LIN {X 0,Y 573.283,Z 141.077,A -85,B 0,C 180,E1 -2348.459,E2 -2348.459} C_VEL
LIN {X 0,Y 573.149,Z 141.164,A -85,B 0,C 180,E1 -2350.598,E2 -2350.598} C_VEL
LIN {X 0,Y 573.117,Z 144.62,A -85,B 0,C 180,E1 -2353.473,E2 -2353.473} C_VEL
LIN {X 0,Y 573.106,Z 148.053,A -85,B 0,C 180,E1 -2356.382,E2 -2356.382} C_VEL
LIN {X 0,Y 573.053,Z 151.315,A -85,B 0,C 180,E1 -2359.206,E2 -2359.206} C_VEL
LIN {X 0,Y 573.008,Z 154.185,A -85,B 0,C 180,E1 -2361.589,E2 -2361.589} C_VEL
LIN {X 0,Y 572.973,Z 157.111,A -85,B 0,C 180,E1 -2364.257,E2 -2364.257} C_VEL
LIN {X 0,Y 572.315,Z 157.815,A -85,B 0,C 180,E1 -2364.839,E2 -2364.839} C_VEL
LIN {X 0,Y 569.431,Z 159.133,A -85,B 0,C 180,E1 -2365.781,E2 -2365.781} C_VEL
LIN {X 0,Y 566.994,Z 160.207,A -85,B 0,C 180,E1 -2366.539,E2 -2366.539} C_VEL
LIN {X 0,Y 565.964,Z 160.962,A -85,B 0,C 180,E1 -2367.126,E2 -2367.126} C_VEL
LIN {X 0,Y 565.89,Z 161.194,A -85,B 0,C 180,E1 -2367.324,E2 -2367.324} C_VEL
LIN {X 0,Y 565.87,Z 164.215,A -85,B 0,C 180,E1 -2369.788,E2 -2369.788} C_VEL
LIN {X 0,Y 565.856,Z 167.674,A -85,B 0,C 180,E1 -2372.426,E2 -2372.426} C_VEL
LIN {X 0,Y 566.893,Z 175.191,A -85,B 0,C 180,E1 -2372.627,E2 -2372.627} C_VEL
LIN {X 0,Y 566.781,Z 187.823,A -85,B 0,C 180,E1 -2373.014,E2 -2373.014} C_VEL
LIN {X 0,Y 566.62,Z 199.261,A -85,B 0,C 180,E1 -2373.5,E2 -2373.5} C_VEL
LIN {X 0,Y 566.449,Z 210.991,A -85,B 0,C 180,E1 -2374.154,E2 -2374.154} C_VEL
LIN {X 0,Y 566.378,Z 222.253,A -85,B 0,C 180,E1 -2374.95,E2 -2374.95} C_VEL
LIN {X 0,Y 566.268,Z 230.723,A -85,B 0,C 180,E1 -2375.684,E2 -2375.684} C_VEL
LIN {X 0,Y 566.138,Z 239.28,A -85,B 0,C 180,E1 -2376.574,E2 -2376.574} C_VEL
LIN {X 0,Y 566.049,Z 247.98,A -85,B 0,C 180,E1 -2377.696,E2 -2377.696} C_VEL
LIN {X 0,Y 565.981,Z 255.315,A -85,B 0,C 180,E1 -2378.885,E2 -2378.885} C_VEL
LIN {X 0,Y 565.935,Z 260.327,A -85,B 0,C 180,E1 -2379.914,E2 -2379.914} C_VEL
LIN {X 0,Y 565.904,Z 264.999,A -85,B 0,C 180,E1 -2381.163,E2 -2381.163} C_VEL
LIN {X 0,Y 565.919,Z 267.606,A -85,B 0,C 180,E1 -2382.114,E2 -2382.114} C_VEL
LIN {X 0,Y 565.855,Z 269.477,A -85,B 0,C 180,E1 -2383.086,E2 -2383.086} C_VEL
LIN {X 0,Y 565.851,Z 270.609,A -85,B 0,C 180,E1 -2384.069,E2 -2384.069} C_VEL
LIN {X 0,Y 565.831,Z 270.999,A -85,B 0,C 180,E1 -2385.07,E2 -2385.07} C_VEL
LIN {X 0,Y 565.849,Z 270.565,A -85,B 0,C 180,E1 -2386.085,E2 -2386.085} C_VEL
LIN {X 0,Y 565.857,Z 269.292,A -85,B 0,C 180,E1 -2387.12,E2 -2387.12} C_VEL
LIN {X 0,Y 565.914,Z 267.122,A -85,B 0,C 180,E1 -2388.17,E2 -2388.17} C_VEL
LIN {X 0,Y 565.918,Z 263.923,A -85,B 0,C 180,E1 -2389.247,E2 -2389.247} C_VEL
LIN {X 0,Y 565.967,Z 259.569,A -85,B 0,C 180,E1 -2390.344,E2 -2390.344} C_VEL
LIN {X 0,Y 565.99,Z 253.825,A -85,B 0,C 180,E1 -2391.469,E2 -2391.469} C_VEL
LIN {X 0,Y 566.059,Z 246.426,A -85,B 0,C 180,E1 -2392.617,E2 -2392.617} C_VEL
LIN {X 0,Y 566.167,Z 238.204,A -85,B 0,C 180,E1 -2393.635,E2 -2393.635} C_VEL
LIN {X 0,Y 566.288,Z 229.712,A -85,B 0,C 180,E1 -2394.499,E2 -2394.499} C_VEL
LIN {X 0,Y 566.367,Z 220.17,A -85,B 0,C 180,E1 -2395.301,E2 -2395.301} C_VEL
LIN {X 0,Y 566.511,Z 208.941,A -85,B 0,C 180,E1 -2396.064,E2 -2396.064} C_VEL
LIN {X 0,Y 566.621,Z 197.802,A -85,B 0,C 180,E1 -2396.659,E2 -2396.659} C_VEL
LIN {X 0,Y 566.796,Z 186.076,A -85,B 0,C 180,E1 -2397.137,E2 -2397.137} C_VEL
LIN {X 0,Y 566.771,Z 173.284,A -85,B 0,C 180,E1 -2397.514,E2 -2397.514} C_VEL
LIN {X 0,Y 565.851,Z 167.7,A -85,B 0,C 180,E1 -2397.652,E2 -2397.652} C_VEL
LIN {X 0,Y 565.875,Z 164.107,A -85,B 0,C 180,E1 -2400.386,E2 -2400.386} C_VEL
LIN {X 0,Y 565.899,Z 160.384,A -85,B 0,C 180,E1 -2403.402,E2 -2403.402} C_VEL
LIN {X 0,Y 565.889,Z 157.605,A -85,B 0,C 180,E1 -2405.805,E2 -2405.805} C_VEL
LIN {X 0,Y 565.923,Z 154.307,A -85,B 0,C 180,E1 -2408.652,E2 -2408.652} C_VEL
LIN {X 0,Y 565.967,Z 151.289,A -85,B 0,C 180,E1 -2411.164,E2 -2411.164} C_VEL
LIN {X 0,Y 566.017,Z 148.71,A -85,B 0,C 180,E1 -2413.406,E2 -2413.406} C_VEL
LIN {X 0,Y 566.011,Z 145.176,A -85,B 0,C 180,E1 -2416.354,E2 -2416.354} C_VEL
LIN {X 0,Y 566.106,Z 142.346,A -85,B 0,C 180,E1 -2418.739,E2 -2418.739} C_VEL
LIN {X 0,Y 566.08,Z 141.976,A -85,B 0,C 180,E1 -2419.267,E2 -2419.267} C_VEL
LIN {X 0,Y 566.22,Z 141.957,A -85,B 0,C 180,E1 -2421.434,E2 -2421.434} C_VEL
LIN {X 0,Y 566.26,Z 141.951,A -85,B 0,C 180,E1 -2424.302,E2 -2424.302} C_VEL
LIN {X 0,Y 566.284,Z 141.948,A -85,B 0,C 180,E1 -2427.866,E2 -2427.866} C_VEL
LIN {X 0,Y 566.296,Z 141.946,A -85,B 0,C 180,E1 -2430.711,E2 -2430.711} C_VEL
LIN {X 0,Y 566.268,Z 141.949,A -85,B 0,C 180,E1 -2432.845,E2 -2432.845} C_VEL
LIN {X 0,Y 566.258,Z 141.951,A -85,B 0,C 180,E1 -2435.698,E2 -2435.698} C_VEL
LIN {X 0,Y 566.226,Z 141.956,A -85,B 0,C 180,E1 -2438.566,E2 -2438.566} C_VEL
LIN {X 0,Y 566.239,Z 141.953,A -85,B 0,C 180,E1 -2441.454,E2 -2441.454} C_VEL
LIN {X 0,Y 566.232,Z 141.956,A -85,B 0,C 180,E1 -2444.507,E2 -2444.507} C_VEL
LIN {X 0,Y 566.2,Z 141.958,A -85,B 0,C 180,E1 -2447.332,E2 -2447.332} C_VEL
LIN {X 0,Y 566.212,Z 141.958,A -85,B 0,C 180,E1 -2450.337,E2 -2450.337} C_VEL
LIN {X 0,Y 566.188,Z 141.959,A -85,B 0,C 180,E1 -2453.404,E2 -2453.404} C_VEL
LIN {X 0,Y 566.21,Z 141.957,A -85,B 0,C 180,E1 -2455.749,E2 -2455.749} C_VEL
LIN {X 0,Y 566.2,Z 141.957,A -85,B 0,C 180,E1 -2458.202,E2 -2458.202} C_VEL
LIN {X 0,Y 566.191,Z 141.96,A -85,B 0,C 180,E1 -2461.077,E2 -2461.077} C_VEL
LIN {X 0,Y 566.209,Z 141.96,A -85,B 0,C 180,E1 -2463.734,E2 -2463.734} C_VEL
LIN {X 0,Y 566.197,Z 141.958,A -85,B 0,C 180,E1 -2466.57,E2 -2466.57} C_VEL
LIN {X 0,Y 566.221,Z 141.955,A -85,B 0,C 180,E1 -2469.273,E2 -2469.273} C_VEL
LIN {X 0,Y 566.209,Z 141.959,A -85,B 0,C 180,E1 -2472.088,E2 -2472.088} C_VEL
LIN {X 0,Y 566.171,Z 141.962,A -85,B 0,C 180,E1 -2475.036,E2 -2475.036} C_VEL
LIN {X 0,Y 566.187,Z 141.96,A -85,B 0,C 180,E1 -2477.911,E2 -2477.911} C_VEL
LIN {X 0,Y 566.216,Z 141.959,A -85,B 0,C 180,E1 -2480.727,E2 -2480.727} C_VEL
LIN {X 0,Y 566.2,Z 141.957,A -85,B 0,C 180,E1 -2483.786,E2 -2483.786} C_VEL
LIN {X 0,Y 566.197,Z 141.958,A -85,B 0,C 180,E1 -2486.268,E2 -2486.268} C_VEL
LIN {X 0,Y 566.193,Z 141.96,A -85,B 0,C 180,E1 -2488.924,E2 -2488.924} C_VEL
LIN {X 0,Y 566.211,Z 141.957,A -85,B 0,C 180,E1 -2491.858,E2 -2491.858} C_VEL
LIN {X 0,Y 566.214,Z 141.957,A -85,B 0,C 180,E1 -2494.251,E2 -2494.251} C_VEL
LIN {X 0,Y 566.171,Z 141.962,A -85,B 0,C 180,E1 -2496.719,E2 -2496.719} C_VEL
LIN {X 0,Y 566.212,Z 141.956,A -85,B 0,C 180,E1 -2499.663,E2 -2499.663} C_VEL
LIN {X 0,Y 566.197,Z 141.959,A -85,B 0,C 180,E1 -2502.669,E2 -2502.669} C_VEL
LIN {X 0,Y 566.222,Z 141.955,A -85,B 0,C 180,E1 -2505.627,E2 -2505.627} C_VEL
LIN {X 0,Y 566.236,Z 141.954,A -85,B 0,C 180,E1 -2508.676,E2 -2508.676} C_VEL
LIN {X 0,Y 566.208,Z 141.956,A -85,B 0,C 180,E1 -2511.434,E2 -2511.434} C_VEL
LIN {X 0,Y 566.26,Z 141.952,A -85,B 0,C 180,E1 -2514.302,E2 -2514.302} C_VEL
LIN {X 0,Y 566.285,Z 141.948,A -85,B 0,C 180,E1 -2517.867,E2 -2517.867} C_VEL
LIN {X 0,Y 566.303,Z 141.946,A -85,B 0,C 180,E1 -2520.711,E2 -2520.711} C_VEL
LIN {X 0,Y 566.272,Z 141.952,A -85,B 0,C 180,E1 -2522.846,E2 -2522.846} C_VEL
LIN {X 0,Y 566.264,Z 141.95,A -85,B 0,C 180,E1 -2525.699,E2 -2525.699} C_VEL
LIN {X 0,Y 566.208,Z 141.957,A -85,B 0,C 180,E1 -2528.566,E2 -2528.566} C_VEL
LIN {X 0,Y 566.245,Z 141.955,A -85,B 0,C 180,E1 -2531.455,E2 -2531.455} C_VEL
LIN {X 0,Y 566.225,Z 141.954,A -85,B 0,C 180,E1 -2534.502,E2 -2534.502} C_VEL
LIN {X 0,Y 566.202,Z 141.96,A -85,B 0,C 180,E1 -2537.332,E2 -2537.332} C_VEL
LIN {X 0,Y 566.208,Z 141.956,A -85,B 0,C 180,E1 -2540.338,E2 -2540.338} C_VEL
LIN {X 0,Y 566.169,Z 141.963,A -85,B 0,C 180,E1 -2543.28,E2 -2543.28} C_VEL
LIN {X 0,Y 566.217,Z 141.958,A -85,B 0,C 180,E1 -2545.749,E2 -2545.749} C_VEL
LIN {X 0,Y 566.206,Z 141.96,A -85,B 0,C 180,E1 -2548.202,E2 -2548.202} C_VEL
LIN {X 0,Y 566.195,Z 141.959,A -85,B 0,C 180,E1 -2551.077,E2 -2551.077} C_VEL
LIN {X 0,Y 566.199,Z 141.958,A -85,B 0,C 180,E1 -2553.732,E2 -2553.732} C_VEL
LIN {X 0,Y 566.202,Z 141.959,A -85,B 0,C 180,E1 -2556.57,E2 -2556.57} C_VEL
LIN {X 0,Y 566.216,Z 141.955,A -85,B 0,C 180,E1 -2559.686,E2 -2559.686} C_VEL
LIN {X 0,Y 566.204,Z 141.958,A -85,B 0,C 180,E1 -2562.917,E2 -2562.917} C_VEL
LIN {X 0,Y 566.197,Z 141.957,A -85,B 0,C 180,E1 -2566.049,E2 -2566.049} C_VEL
LIN {X 0,Y 566.206,Z 141.957,A -85,B 0,C 180,E1 -2569.215,E2 -2569.215} C_VEL
LIN {X 0,Y 566.188,Z 141.961,A -85,B 0,C 180,E1 -2571.637,E2 -2571.637} C_VEL
LIN {X 0,Y 566.237,Z 141.963,A -85,B 0,C 180,E1 -2572.989,E2 -2572.989} C_VEL
LIN {X 0,Y 566.793,Z 145.917,A -85,B 0,C 180,E1 -2574.354,E2 -2574.354} C_VEL
LIN {X 0,Y 566.8,Z 152.68,A -85,B 0,C 180,E1 -2576.557,E2 -2576.557} C_VEL
LIN {X 0,Y 566.62,Z 161.803,A -85,B 0,C 180,E1 -2579.433,E2 -2579.433} C_VEL
LIN {X 0,Y 566.518,Z 171.071,A -85,B 0,C 180,E1 -2582.276,E2 -2582.276} C_VEL
LIN {X 0,Y 566.418,Z 180.338,A -85,B 0,C 180,E1 -2585.048,E2 -2585.048} C_VEL
LIN {X 0,Y 566.323,Z 190.929,A -85,B 0,C 180,E1 -2588.143,E2 -2588.143} C_VEL
LIN {X 0,Y 566.186,Z 201.521,A -85,B 0,C 180,E1 -2591.172,E2 -2591.172} C_VEL
LIN {X 0,Y 566.112,Z 212.112,A -85,B 0,C 180,E1 -2594.15,E2 -2594.15} C_VEL
LIN {X 0,Y 566.003,Z 222.703,A -85,B 0,C 180,E1 -2597.085,E2 -2597.085} C_VEL
LIN {X 0,Y 566.011,Z 223.53,A -85,B 0,C 180,E1 -2597.313,E2 -2597.313} C_VEL
LIN {X 0,Y 566.93,Z 230.375,A -85,B 0,C 180,E1 -2597.471,E2 -2597.471} C_VEL
LIN {X 0,Y 566.839,Z 242.5,A -85,B 0,C 180,E1 -2597.787,E2 -2597.787} C_VEL
LIN {X 0,Y 566.68,Z 254.321,A -85,B 0,C 180,E1 -2598.228,E2 -2598.228} C_VEL
LIN {X 0,Y 566.532,Z 266.981,A -85,B 0,C 180,E1 -2598.868,E2 -2598.868} C_VEL
LIN {X 0,Y 566.434,Z 278.748,A -85,B 0,C 180,E1 -2599.636,E2 -2599.636} C_VEL
LIN {X 0,Y 566.301,Z 287.648,A -85,B 0,C 180,E1 -2600.355,E2 -2600.355} C_VEL
LIN {X 0,Y 566.166,Z 296.788,A -85,B 0,C 180,E1 -2601.254,E2 -2601.254} C_VEL
LIN {X 0,Y 566.081,Z 305.691,A -85,B 0,C 180,E1 -2602.33,E2 -2602.33} C_VEL
LIN {X 0,Y 565.968,Z 312.956,A -85,B 0,C 180,E1 -2603.422,E2 -2603.422} C_VEL
LIN {X 0,Y 566.004,Z 317.681,A -85,B 0,C 180,E1 -2604.299,E2 -2604.299} C_VEL
LIN {X 0,Y 565.933,Z 322.372,A -85,B 0,C 180,E1 -2605.37,E2 -2605.37} C_VEL
LIN {X 0,Y 565.927,Z 325.957,A -85,B 0,C 180,E1 -2606.44,E2 -2606.44} C_VEL
LIN {X 0,Y 565.878,Z 327.809,A -85,B 0,C 180,E1 -2607.153,E2 -2607.153} C_VEL
LIN {X 0,Y 565.841,Z 329.2,A -85,B 0,C 180,E1 -2607.865,E2 -2607.865} C_VEL
LIN {X 0,Y 565.841,Z 330.784,A -85,B 0,C 180,E1 -2609.288,E2 -2609.288} C_VEL
LIN {X 0,Y 565.839,Z 331,A -85,B 0,C 180,E1 -2610,E2 -2610} C_VEL
LIN {X 0,Y 565.846,Z 330.185,A -85,B 0,C 180,E1 -2611.424,E2 -2611.424} C_VEL
LIN {X 0,Y 565.841,Z 329.201,A -85,B 0,C 180,E1 -2612.136,E2 -2612.136} C_VEL
LIN {X 0,Y 565.878,Z 327.809,A -85,B 0,C 180,E1 -2612.848,E2 -2612.848} C_VEL
LIN {X 0,Y 565.926,Z 324.896,A -85,B 0,C 180,E1 -2613.917,E2 -2613.917} C_VEL
LIN {X 0,Y 565.878,Z 320.949,A -85,B 0,C 180,E1 -2614.988,E2 -2614.988} C_VEL
LIN {X 0,Y 566.002,Z 315.866,A -85,B 0,C 180,E1 -2616.059,E2 -2616.059} C_VEL
LIN {X 0,Y 566.041,Z 309.469,A -85,B 0,C 180,E1 -2617.132,E2 -2617.132} C_VEL
LIN {X 0,Y 566.134,Z 301.477,A -85,B 0,C 180,E1 -2618.208,E2 -2618.208} C_VEL
LIN {X 0,Y 566.229,Z 293.335,A -85,B 0,C 180,E1 -2619.106,E2 -2619.106} C_VEL
LIN {X 0,Y 566.344,Z 283.4,A -85,B 0,C 180,E1 -2620.005,E2 -2620.005} C_VEL
LIN {X 0,Y 566.501,Z 272.326,A -85,B 0,C 180,E1 -2620.805,E2 -2620.805} C_VEL
LIN {X 0,Y 566.574,Z 261.175,A -85,B 0,C 180,E1 -2621.448,E2 -2621.448} C_VEL
LIN {X 0,Y 566.741,Z 248.985,A -85,B 0,C 180,E1 -2621.988,E2 -2621.988} C_VEL
LIN {X 0,Y 566.918,Z 236.171,A -85,B 0,C 180,E1 -2622.393,E2 -2622.393} C_VEL
LIN {X 0,Y 566.73,Z 228.079,A -85,B 0,C 180,E1 -2622.58,E2 -2622.58} C_VEL
LIN {X 0,Y 566.011,Z 223.53,A -85,B 0,C 180,E1 -2622.687,E2 -2622.687} C_VEL
LIN {X 0,Y 566.087,Z 213.435,A -85,B 0,C 180,E1 -2625.481,E2 -2625.481} C_VEL
LIN {X 0,Y 566.167,Z 202.844,A -85,B 0,C 180,E1 -2628.454,E2 -2628.454} C_VEL
LIN {X 0,Y 566.246,Z 193.576,A -85,B 0,C 180,E1 -2631.096,E2 -2631.096} C_VEL
LIN {X 0,Y 566.365,Z 184.309,A -85,B 0,C 180,E1 -2633.784,E2 -2633.784} C_VEL
LIN {X 0,Y 566.485,Z 175.042,A -85,B 0,C 180,E1 -2636.528,E2 -2636.528} C_VEL
LIN {X 0,Y 566.553,Z 165.774,A -85,B 0,C 180,E1 -2639.34,E2 -2639.34} C_VEL
LIN {X 0,Y 566.704,Z 156.507,A -85,B 0,C 180,E1 -2642.227,E2 -2642.227} C_VEL
LIN {X 0,Y 566.837,Z 148.564,A -85,B 0,C 180,E1 -2644.774,E2 -2644.774} C_VEL
LIN {X 0,Y 566.568,Z 144.069,A -85,B 0,C 180,E1 -2646.264,E2 -2646.264} C_VEL
LIN {X 0,Y 566.239,Z 141.957,A -85,B 0,C 180,E1 -2647.011,E2 -2647.011} C_VEL
LIN {X 0,Y 566.22,Z 141.957,A -85,B 0,C 180,E1 -2649.686,E2 -2649.686} C_VEL
LIN {X 0,Y 566.216,Z 141.959,A -85,B 0,C 180,E1 -2652.088,E2 -2652.088} C_VEL
LIN {X 0,Y 566.178,Z 141.963,A -85,B 0,C 180,E1 -2655.036,E2 -2655.036} C_VEL
LIN {X 0,Y 566.194,Z 141.961,A -85,B 0,C 180,E1 -2657.91,E2 -2657.91} C_VEL
LIN {X 0,Y 566.225,Z 141.956,A -85,B 0,C 180,E1 -2660.727,E2 -2660.727} C_VEL
LIN {X 0,Y 566.19,Z 141.96,A -85,B 0,C 180,E1 -2663.788,E2 -2663.788} C_VEL
LIN {X 0,Y 566.217,Z 141.958,A -85,B 0,C 180,E1 -2666.266,E2 -2666.266} C_VEL
LIN {X 0,Y 566.199,Z 141.959,A -85,B 0,C 180,E1 -2668.923,E2 -2668.923} C_VEL
LIN {X 0,Y 566.217,Z 141.957,A -85,B 0,C 180,E1 -2671.857,E2 -2671.857} C_VEL
LIN {X 0,Y 566.219,Z 141.957,A -85,B 0,C 180,E1 -2674.251,E2 -2674.251} C_VEL
LIN {X 0,Y 566.176,Z 141.962,A -85,B 0,C 180,E1 -2676.719,E2 -2676.719} C_VEL
LIN {X 0,Y 566.212,Z 141.958,A -85,B 0,C 180,E1 -2679.662,E2 -2679.662} C_VEL
LIN {X 0,Y 566.204,Z 141.959,A -85,B 0,C 180,E1 -2682.668,E2 -2682.668} C_VEL
LIN {X 0,Y 566.24,Z 141.955,A -85,B 0,C 180,E1 -2685.627,E2 -2685.627} C_VEL
LIN {X 0,Y 566.24,Z 141.955,A -85,B 0,C 180,E1 -2688.675,E2 -2688.675} C_VEL
LIN {X 0,Y 566.233,Z 141.956,A -85,B 0,C 180,E1 -2691.434,E2 -2691.434} C_VEL
LIN {X 0,Y 566.265,Z 141.951,A -85,B 0,C 180,E1 -2694.301,E2 -2694.301} C_VEL
LIN {X 0,Y 566.288,Z 141.949,A -85,B 0,C 180,E1 -2697.866,E2 -2697.866} C_VEL
LIN {X 0,Y 566.308,Z 141.947,A -85,B 0,C 180,E1 -2700.711,E2 -2700.711} C_VEL
LIN {X 0,Y 566.276,Z 141.951,A -85,B 0,C 180,E1 -2702.845,E2 -2702.845} C_VEL
LIN {X 0,Y 566.26,Z 141.954,A -85,B 0,C 180,E1 -2705.698,E2 -2705.698} C_VEL
LIN {X 0,Y 566.225,Z 141.957,A -85,B 0,C 180,E1 -2708.565,E2 -2708.565} C_VEL
LIN {X 0,Y 566.082,Z 142.035,A -85,B 0,C 180,E1 -2710.732,E2 -2710.732} C_VEL
LIN {X 0,Y 566.051,Z 145.513,A -85,B 0,C 180,E1 -2713.644,E2 -2713.644} C_VEL
LIN {X 0,Y 566.047,Z 148.957,A -85,B 0,C 180,E1 -2716.592,E2 -2716.592} C_VEL
LIN {X 0,Y 565.936,Z 152.413,A -85,B 0,C 180,E1 -2719.59,E2 -2719.59} C_VEL
LIN {X 0,Y 565.916,Z 155.096,A -85,B 0,C 180,E1 -2721.873,E2 -2721.873} C_VEL
LIN {X 0,Y 565.903,Z 157.781,A -85,B 0,C 180,E1 -2724.248,E2 -2724.248} C_VEL
LIN {X 0,Y 565.903,Z 160.372,A -85,B 0,C 180,E1 -2726.597,E2 -2726.597} C_VEL
LIN {X 0,Y 565.89,Z 161.194,A -85,B 0,C 180,E1 -2727.324,E2 -2727.324} C_VEL
LIN {X 0,Y 565.244,Z 161.922,A -85,B 0,C 180,E1 -2727.914,E2 -2727.914} C_VEL
LIN {X 0,Y 562.374,Z 163.269,A -85,B 0,C 180,E1 -2728.869,E2 -2728.869} C_VEL
LIN {X 0,Y 559.925,Z 164.365,A -85,B 0,C 180,E1 -2729.637,E2 -2729.637} C_VEL
LIN {X 0,Y 558.86,Z 165.144,A -85,B 0,C 180,E1 -2730.231,E2 -2730.231} C_VEL
LIN {X 0,Y 558.767,Z 165.387,A -85,B 0,C 180,E1 -2730.433,E2 -2730.433} C_VEL
LIN {X 0,Y 558.759,Z 167.671,A -85,B 0,C 180,E1 -2732.26,E2 -2732.26} C_VEL
LIN {X 0,Y 559.961,Z 175.931,A -85,B 0,C 180,E1 -2732.489,E2 -2732.489} C_VEL
LIN {X 0,Y 559.827,Z 188.735,A -85,B 0,C 180,E1 -2732.897,E2 -2732.897} C_VEL
LIN {X 0,Y 559.621,Z 200.62,A -85,B 0,C 180,E1 -2733.425,E2 -2733.425} C_VEL
LIN {X 0,Y 559.462,Z 212.087,A -85,B 0,C 180,E1 -2734.087,E2 -2734.087} C_VEL
LIN {X 0,Y 559.356,Z 222.83,A -85,B 0,C 180,E1 -2734.867,E2 -2734.867} C_VEL
LIN {X 0,Y 559.206,Z 232.71,A -85,B 0,C 180,E1 -2735.76,E2 -2735.76} C_VEL
LIN {X 0,Y 559.069,Z 241.597,A -85,B 0,C 180,E1 -2736.748,E2 -2736.748} C_VEL
LIN {X 0,Y 558.96,Z 249.3,A -85,B 0,C 180,E1 -2737.797,E2 -2737.797} C_VEL
LIN {X 0,Y 558.896,Z 256.106,A -85,B 0,C 180,E1 -2738.957,E2 -2738.957} C_VEL
LIN {X 0,Y 558.859,Z 260.573,A -85,B 0,C 180,E1 -2739.904,E2 -2739.904} C_VEL
LIN {X 0,Y 558.81,Z 264.676,A -85,B 0,C 180,E1 -2741.009,E2 -2741.009} C_VEL
LIN {X 0,Y 558.82,Z 267.655,A -85,B 0,C 180,E1 -2742.096,E2 -2742.096} C_VEL
LIN {X 0,Y 558.767,Z 269.62,A -85,B 0,C 180,E1 -2743.155,E2 -2743.155} C_VEL
LIN {X 0,Y 558.765,Z 270.703,A -85,B 0,C 180,E1 -2744.198,E2 -2744.198} C_VEL
LIN {X 0,Y 558.75,Z 270.968,A -85,B 0,C 180,E1 -2745.221,E2 -2745.221} C_VEL
LIN {X 0,Y 558.758,Z 270.465,A -85,B 0,C 180,E1 -2746.228,E2 -2746.228} C_VEL
LIN {X 0,Y 558.759,Z 269.178,A -85,B 0,C 180,E1 -2747.218,E2 -2747.218} C_VEL
LIN {X 0,Y 558.815,Z 267.151,A -85,B 0,C 180,E1 -2748.197,E2 -2748.197} C_VEL
LIN {X 0,Y 558.822,Z 264.414,A -85,B 0,C 180,E1 -2749.158,E2 -2749.158} C_VEL
LIN {X 0,Y 558.881,Z 259.874,A -85,B 0,C 180,E1 -2750.343,E2 -2750.343} C_VEL
LIN {X 0,Y 558.925,Z 253.564,A -85,B 0,C 180,E1 -2751.598,E2 -2751.598} C_VEL
LIN {X 0,Y 558.985,Z 246.996,A -85,B 0,C 180,E1 -2752.632,E2 -2752.632} C_VEL
LIN {X 0,Y 559.084,Z 239.797,A -85,B 0,C 180,E1 -2753.563,E2 -2753.563} C_VEL
LIN {X 0,Y 559.262,Z 230.183,A -85,B 0,C 180,E1 -2754.575,E2 -2754.575} C_VEL
LIN {X 0,Y 559.392,Z 219.751,A -85,B 0,C 180,E1 -2755.463,E2 -2755.463} C_VEL
LIN {X 0,Y 559.526,Z 208.818,A -85,B 0,C 180,E1 -2756.211,E2 -2756.211} C_VEL
LIN {X 0,Y 559.687,Z 197.086,A -85,B 0,C 180,E1 -2756.838,E2 -2756.838} C_VEL
LIN {X 0,Y 559.874,Z 184.86,A -85,B 0,C 180,E1 -2757.332,E2 -2757.332} C_VEL
LIN {X 0,Y 559.794,Z 173.908,A -85,B 0,C 180,E1 -2757.656,E2 -2757.656} C_VEL
LIN {X 0,Y 558.763,Z 167.684,A -85,B 0,C 180,E1 -2757.819,E2 -2757.819} C_VEL
LIN {X 0,Y 558.794,Z 164.191,A -85,B 0,C 180,E1 -2760.626,E2 -2760.626} C_VEL
LIN {X 0,Y 558.813,Z 160.368,A -85,B 0,C 180,E1 -2763.884,E2 -2763.884} C_VEL
LIN {X 0,Y 558.833,Z 157.24,A -85,B 0,C 180,E1 -2766.643,E2 -2766.643} C_VEL
LIN {X 0,Y 558.849,Z 153.987,A -85,B 0,C 180,E1 -2769.383,E2 -2769.383} C_VEL
LIN {X 0,Y 558.92,Z 150.432,A -85,B 0,C 180,E1 -2772.435,E2 -2772.435} C_VEL
LIN {X 0,Y 558.972,Z 146.812,A -85,B 0,C 180,E1 -2775.493,E2 -2775.493} C_VEL
LIN {X 0,Y 559.037,Z 143.059,A -85,B 0,C 180,E1 -2778.689,E2 -2778.689} C_VEL
LIN {X 0,Y 559.177,Z 142.834,A -85,B 0,C 180,E1 -2781.325,E2 -2781.325} C_VEL
LIN {X 0,Y 559.228,Z 142.827,A -85,B 0,C 180,E1 -2784.23,E2 -2784.23} C_VEL
LIN {X 0,Y 559.255,Z 142.824,A -85,B 0,C 180,E1 -2787.839,E2 -2787.839} C_VEL
LIN {X 0,Y 559.267,Z 142.821,A -85,B 0,C 180,E1 -2790.72,E2 -2790.72} C_VEL
LIN {X 0,Y 559.234,Z 142.824,A -85,B 0,C 180,E1 -2792.881,E2 -2792.881} C_VEL
LIN {X 0,Y 559.227,Z 142.828,A -85,B 0,C 180,E1 -2795.77,E2 -2795.77} C_VEL
LIN {X 0,Y 559.184,Z 142.832,A -85,B 0,C 180,E1 -2798.674,E2 -2798.674} C_VEL
LIN {X 0,Y 559.203,Z 142.83,A -85,B 0,C 180,E1 -2801.6,E2 -2801.6} C_VEL
LIN {X 0,Y 559.197,Z 142.832,A -85,B 0,C 180,E1 -2804.596,E2 -2804.596} C_VEL
LIN {X 0,Y 559.16,Z 142.835,A -85,B 0,C 180,E1 -2807.557,E2 -2807.557} C_VEL
LIN {X 0,Y 559.168,Z 142.834,A -85,B 0,C 180,E1 -2809.837,E2 -2809.837} C_VEL
LIN {X 0,Y 559.138,Z 142.837,A -85,B 0,C 180,E1 -2812.153,E2 -2812.153} C_VEL
LIN {X 0,Y 559.176,Z 142.834,A -85,B 0,C 180,E1 -2815.187,E2 -2815.187} C_VEL
LIN {X 0,Y 559.178,Z 142.836,A -85,B 0,C 180,E1 -2817.712,E2 -2817.712} C_VEL
LIN {X 0,Y 559.154,Z 142.838,A -85,B 0,C 180,E1 -2820.183,E2 -2820.183} C_VEL
LIN {X 0,Y 559.172,Z 142.835,A -85,B 0,C 180,E1 -2822.714,E2 -2822.714} C_VEL
LIN {X 0,Y 559.125,Z 142.84,A -85,B 0,C 180,E1 -2825.324,E2 -2825.324} C_VEL
LIN {X 0,Y 559.132,Z 142.837,A -85,B 0,C 180,E1 -2828.018,E2 -2828.018} C_VEL
LIN {X 0,Y 559.173,Z 142.834,A -85,B 0,C 180,E1 -2830.811,E2 -2830.811} C_VEL
LIN {X 0,Y 559.139,Z 142.837,A -85,B 0,C 180,E1 -2833.734,E2 -2833.734} C_VEL
LIN {X 0,Y 559.144,Z 142.838,A -85,B 0,C 180,E1 -2836.804,E2 -2836.804} C_VEL
LIN {X 0,Y 559.154,Z 142.837,A -85,B 0,C 180,E1 -2839.188,E2 -2839.188} C_VEL
LIN {X 0,Y 559.134,Z 142.84,A -85,B 0,C 180,E1 -2841.983,E2 -2841.983} C_VEL
LIN {X 0,Y 559.146,Z 142.837,A -85,B 0,C 180,E1 -2844.785,E2 -2844.785} C_VEL
LIN {X 0,Y 559.154,Z 142.835,A -85,B 0,C 180,E1 -2847.365,E2 -2847.365} C_VEL
LIN {X 0,Y 559.145,Z 142.837,A -85,B 0,C 180,E1 -2850.143,E2 -2850.143} C_VEL
LIN {X 0,Y 559.169,Z 142.834,A -85,B 0,C 180,E1 -2853.098,E2 -2853.098} C_VEL
LIN {X 0,Y 559.155,Z 142.835,A -85,B 0,C 180,E1 -2855.495,E2 -2855.495} C_VEL
LIN {X 0,Y 559.173,Z 142.835,A -85,B 0,C 180,E1 -2858.624,E2 -2858.624} C_VEL
LIN {X 0,Y 559.165,Z 142.835,A -85,B 0,C 180,E1 -2860.927,E2 -2860.927} C_VEL
LIN {X 0,Y 559.164,Z 142.835,A -85,B 0,C 180,E1 -2863.948,E2 -2863.948} C_VEL
LIN {X 0,Y 559.166,Z 142.836,A -85,B 0,C 180,E1 -2866.184,E2 -2866.184} C_VEL
LIN {X 0,Y 559.208,Z 142.83,A -85,B 0,C 180,E1 -2868.605,E2 -2868.605} C_VEL
LIN {X 0,Y 559.172,Z 142.833,A -85,B 0,C 180,E1 -2871.326,E2 -2871.326} C_VEL
LIN {X 0,Y 559.23,Z 142.827,A -85,B 0,C 180,E1 -2874.23,E2 -2874.23} C_VEL
LIN {X 0,Y 559.256,Z 142.824,A -85,B 0,C 180,E1 -2877.84,E2 -2877.84} C_VEL
LIN {X 0,Y 559.273,Z 142.821,A -85,B 0,C 180,E1 -2880.72,E2 -2880.72} C_VEL
LIN {X 0,Y 559.239,Z 142.827,A -85,B 0,C 180,E1 -2882.882,E2 -2882.882} C_VEL
LIN {X 0,Y 559.232,Z 142.826,A -85,B 0,C 180,E1 -2885.771,E2 -2885.771} C_VEL
LIN {X 0,Y 559.173,Z 142.834,A -85,B 0,C 180,E1 -2888.675,E2 -2888.675} C_VEL
LIN {X 0,Y 559.209,Z 142.83,A -85,B 0,C 180,E1 -2891.601,E2 -2891.601} C_VEL
LIN {X 0,Y 559.183,Z 142.832,A -85,B 0,C 180,E1 -2894.588,E2 -2894.588} C_VEL
LIN {X 0,Y 559.161,Z 142.837,A -85,B 0,C 180,E1 -2897.557,E2 -2897.557} C_VEL
LIN {X 0,Y 559.168,Z 142.837,A -85,B 0,C 180,E1 -2899.838,E2 -2899.838} C_VEL
LIN {X 0,Y 559.144,Z 142.84,A -85,B 0,C 180,E1 -2902.153,E2 -2902.153} C_VEL
LIN {X 0,Y 559.179,Z 142.832,A -85,B 0,C 180,E1 -2905.298,E2 -2905.298} C_VEL
LIN {X 0,Y 559.16,Z 142.835,A -85,B 0,C 180,E1 -2907.714,E2 -2907.714} C_VEL
LIN {X 0,Y 559.153,Z 142.835,A -85,B 0,C 180,E1 -2910.183,E2 -2910.183} C_VEL
LIN {X 0,Y 559.154,Z 142.835,A -85,B 0,C 180,E1 -2912.716,E2 -2912.716} C_VEL
LIN {X 0,Y 559.13,Z 142.84,A -85,B 0,C 180,E1 -2915.324,E2 -2915.324} C_VEL
LIN {X 0,Y 559.134,Z 142.84,A -85,B 0,C 180,E1 -2918.018,E2 -2918.018} C_VEL
LIN {X 0,Y 559.158,Z 142.835,A -85,B 0,C 180,E1 -2920.813,E2 -2920.813} C_VEL
LIN {X 0,Y 559.144,Z 142.837,A -85,B 0,C 180,E1 -2923.734,E2 -2923.734} C_VEL
LIN {X 0,Y 559.148,Z 142.835,A -85,B 0,C 180,E1 -2926.804,E2 -2926.804} C_VEL
LIN {X 0,Y 559.158,Z 142.836,A -85,B 0,C 180,E1 -2929.188,E2 -2929.188} C_VEL
LIN {X 0,Y 559.135,Z 142.84,A -85,B 0,C 180,E1 -2931.983,E2 -2931.983} C_VEL
LIN {X 0,Y 559.215,Z 143.016,A -85,B 0,C 180,E1 -2932.8,E2 -2932.8} C_VEL
LIN {X 0,Y 559.845,Z 147.254,A -85,B 0,C 180,E1 -2934.287,E2 -2934.287} C_VEL
LIN {X 0,Y 559.794,Z 155.185,A -85,B 0,C 180,E1 -2936.899,E2 -2936.899} C_VEL
LIN {X 0,Y 559.643,Z 164.451,A -85,B 0,C 180,E1 -2939.846,E2 -2939.846} C_VEL
LIN {X 0,Y 559.499,Z 173.719,A -85,B 0,C 180,E1 -2942.711,E2 -2942.711} C_VEL
LIN {X 0,Y 559.378,Z 182.986,A -85,B 0,C 180,E1 -2945.505,E2 -2945.505} C_VEL
LIN {X 0,Y 559.234,Z 193.577,A -85,B 0,C 180,E1 -2948.626,E2 -2948.626} C_VEL
LIN {X 0,Y 559.134,Z 202.844,A -85,B 0,C 180,E1 -2951.306,E2 -2951.306} C_VEL
LIN {X 0,Y 559.052,Z 213.436,A -85,B 0,C 180,E1 -2954.319,E2 -2954.319} C_VEL
LIN {X 0,Y 558.938,Z 223.53,A -85,B 0,C 180,E1 -2957.15,E2 -2957.15} C_VEL
LIN {X 0,Y 560.018,Z 231.514,A -85,B 0,C 180,E1 -2957.337,E2 -2957.337} C_VEL
LIN {X 0,Y 559.899,Z 243.88,A -85,B 0,C 180,E1 -2957.679,E2 -2957.679} C_VEL
LIN {X 0,Y 559.718,Z 256.284,A -85,B 0,C 180,E1 -2958.171,E2 -2958.171} C_VEL
LIN {X 0,Y 559.555,Z 267.767,A -85,B 0,C 180,E1 -2958.773,E2 -2958.773} C_VEL
LIN {X 0,Y 559.424,Z 278.748,A -85,B 0,C 180,E1 -2959.504,E2 -2959.504} C_VEL
LIN {X 0,Y 559.244,Z 289.602,A -85,B 0,C 180,E1 -2960.415,E2 -2960.415} C_VEL
LIN {X 0,Y 559.127,Z 298.414,A -85,B 0,C 180,E1 -2961.325,E2 -2961.325} C_VEL
LIN {X 0,Y 558.996,Z 307.001,A -85,B 0,C 180,E1 -2962.414,E2 -2962.414} C_VEL
LIN {X 0,Y 558.885,Z 314.689,A -85,B 0,C 180,E1 -2963.649,E2 -2963.649} C_VEL
LIN {X 0,Y 558.869,Z 319.366,A -85,B 0,C 180,E1 -2964.588,E2 -2964.588} C_VEL
LIN {X 0,Y 558.869,Z 323.678,A -85,B 0,C 180,E1 -2965.673,E2 -2965.673} C_VEL
LIN {X 0,Y 558.836,Z 325.957,A -85,B 0,C 180,E1 -2966.395,E2 -2966.395} C_VEL
LIN {X 0,Y 558.799,Z 327.809,A -85,B 0,C 180,E1 -2967.116,E2 -2967.116} C_VEL
LIN {X 0,Y 558.747,Z 329.2,A -85,B 0,C 180,E1 -2967.838,E2 -2967.838} C_VEL
LIN {X 0,Y 558.741,Z 330.785,A -85,B 0,C 180,E1 -2969.279,E2 -2969.279} C_VEL
LIN {X 0,Y 558.74,Z 331,A -85,B 0,C 180,E1 -2970,E2 -2970} C_VEL
LIN {X 0,Y 558.745,Z 330.185,A -85,B 0,C 180,E1 -2971.442,E2 -2971.442} C_VEL
LIN {X 0,Y 558.747,Z 329.2,A -85,B 0,C 180,E1 -2972.163,E2 -2972.163} C_VEL
LIN {X 0,Y 558.799,Z 327.809,A -85,B 0,C 180,E1 -2972.884,E2 -2972.884} C_VEL
LIN {X 0,Y 558.844,Z 324.895,A -85,B 0,C 180,E1 -2973.966,E2 -2973.966} C_VEL
LIN {X 0,Y 558.798,Z 320.949,A -85,B 0,C 180,E1 -2975.051,E2 -2975.051} C_VEL
LIN {X 0,Y 558.922,Z 315.866,A -85,B 0,C 180,E1 -2976.136,E2 -2976.136} C_VEL
LIN {X 0,Y 558.978,Z 309.468,A -85,B 0,C 180,E1 -2977.223,E2 -2977.223} C_VEL
LIN {X 0,Y 559.099,Z 301.477,A -85,B 0,C 180,E1 -2978.312,E2 -2978.312} C_VEL
LIN {X 0,Y 559.195,Z 293.335,A -85,B 0,C 180,E1 -2979.221,E2 -2979.221} C_VEL
LIN {X 0,Y 559.358,Z 283.4,A -85,B 0,C 180,E1 -2980.131,E2 -2980.131} C_VEL
LIN {X 0,Y 559.511,Z 272.435,A -85,B 0,C 180,E1 -2980.935,E2 -2980.935} C_VEL
LIN {X 0,Y 559.637,Z 260.82,A -85,B 0,C 180,E1 -2981.61,E2 -2981.61} C_VEL
LIN {X 0,Y 559.816,Z 248.984,A -85,B 0,C 180,E1 -2982.139,E2 -2982.139} C_VEL
LIN {X 0,Y 559.989,Z 236.171,A -85,B 0,C 180,E1 -2982.549,E2 -2982.549} C_VEL
LIN {X 0,Y 559.814,Z 228.936,A -85,B 0,C 180,E1 -2982.72,E2 -2982.72} C_VEL
LIN {X 0,Y 558.938,Z 223.53,A -85,B 0,C 180,E1 -2982.85,E2 -2982.85} C_VEL
LIN {X 0,Y 559.052,Z 213.435,A -85,B 0,C 180,E1 -2985.681,E2 -2985.681} C_VEL
LIN {X 0,Y 559.134,Z 202.844,A -85,B 0,C 180,E1 -2988.695,E2 -2988.695} C_VEL
LIN {X 0,Y 559.228,Z 192.915,A -85,B 0,C 180,E1 -2991.567,E2 -2991.567} C_VEL
LIN {X 0,Y 559.378,Z 182.985,A -85,B 0,C 180,E1 -2994.495,E2 -2994.495} C_VEL
LIN {X 0,Y 559.5,Z 173.718,A -85,B 0,C 180,E1 -2997.29,E2 -2997.29} C_VEL
LIN {X 0,Y 559.644,Z 164.45,A -85,B 0,C 180,E1 -3000.154,E2 -3000.154} C_VEL
LIN {X 0,Y 559.795,Z 155.184,A -85,B 0,C 180,E1 -3003.101,E2 -3003.101} C_VEL
LIN {X 0,Y 559.853,Z 147.183,A -85,B 0,C 180,E1 -3005.713,E2 -3005.713} C_VEL
LIN {X 0,Y 559.175,Z 142.836,A -85,B 0,C 180,E1 -3007.302,E2 -3007.302} C_VEL
LIN {X 0,Y 559.165,Z 142.836,A -85,B 0,C 180,E1 -3009.942,E2 -3009.942} C_VEL
LIN {X 0,Y 559.166,Z 142.835,A -85,B 0,C 180,E1 -3012.743,E2 -3012.743} C_VEL
LIN {X 0,Y 559.158,Z 142.836,A -85,B 0,C 180,E1 -3015.761,E2 -3015.761} C_VEL
LIN {X 0,Y 559.17,Z 142.837,A -85,B 0,C 180,E1 -3018.23,E2 -3018.23} C_VEL
LIN {X 0,Y 559.181,Z 142.835,A -85,B 0,C 180,E1 -3021.191,E2 -3021.191} C_VEL
LIN {X 0,Y 559.145,Z 142.837,A -85,B 0,C 180,E1 -3023.789,E2 -3023.789} C_VEL
LIN {X 0,Y 559.171,Z 142.836,A -85,B 0,C 180,E1 -3026.425,E2 -3026.425} C_VEL
LIN {X 0,Y 559.163,Z 142.835,A -85,B 0,C 180,E1 -3028.981,E2 -3028.981} C_VEL
LIN {X 0,Y 559.173,Z 142.835,A -85,B 0,C 180,E1 -3031.619,E2 -3031.619} C_VEL
LIN {X 0,Y 559.186,Z 142.832,A -85,B 0,C 180,E1 -3033.903,E2 -3033.903} C_VEL
LIN {X 0,Y 559.146,Z 142.839,A -85,B 0,C 180,E1 -3036.571,E2 -3036.571} C_VEL
LIN {X 0,Y 559.181,Z 142.835,A -85,B 0,C 180,E1 -3039.395,E2 -3039.395} C_VEL
LIN {X 0,Y 559.146,Z 142.837,A -85,B 0,C 180,E1 -3041.685,E2 -3041.685} C_VEL
LIN {X 0,Y 559.167,Z 142.835,A -85,B 0,C 180,E1 -3043.948,E2 -3043.948} C_VEL
LIN {X 0,Y 559.176,Z 142.834,A -85,B 0,C 180,E1 -3046.184,E2 -3046.184} C_VEL
LIN {X 0,Y 559.2,Z 142.831,A -85,B 0,C 180,E1 -3049.133,E2 -3049.133} C_VEL
LIN {X 0,Y 559.209,Z 142.829,A -85,B 0,C 180,E1 -3052.053,E2 -3052.053} C_VEL
LIN {X 0,Y 559.257,Z 142.824,A -85,B 0,C 180,E1 -3054.953,E2 -3054.953} C_VEL
LIN {X 0,Y 559.259,Z 142.824,A -85,B 0,C 180,E1 -3057.839,E2 -3057.839} C_VEL
LIN {X 0,Y 559.278,Z 142.823,A -85,B 0,C 180,E1 -3060.72,E2 -3060.72} C_VEL
LIN {X 0,Y 559.242,Z 142.827,A -85,B 0,C 180,E1 -3062.881,E2 -3062.881} C_VEL
LIN {X 0,Y 559.229,Z 142.83,A -85,B 0,C 180,E1 -3065.77,E2 -3065.77} C_VEL
LIN {X 0,Y 559.182,Z 142.835,A -85,B 0,C 180,E1 -3068.674,E2 -3068.674} C_VEL
LIN {X 0,Y 559.024,Z 142.927,A -85,B 0,C 180,E1 -3070.869,E2 -3070.869} C_VEL
LIN {X 0,Y 559,Z 146.396,A -85,B 0,C 180,E1 -3073.82,E2 -3073.82} C_VEL
LIN {X 0,Y 558.971,Z 149.87,A -85,B 0,C 180,E1 -3076.809,E2 -3076.809} C_VEL
LIN {X 0,Y 558.871,Z 153.354,A -85,B 0,C 180,E1 -3079.848,E2 -3079.848} C_VEL
LIN {X 0,Y 558.828,Z 156.008,A -85,B 0,C 180,E1 -3082.165,E2 -3082.165} C_VEL
LIN {X 0,Y 558.835,Z 158.752,A -85,B 0,C 180,E1 -3084.52,E2 -3084.52} C_VEL
LIN {X 0,Y 558.803,Z 161.82,A -85,B 0,C 180,E1 -3087.313,E2 -3087.313} C_VEL
LIN {X 0,Y 558.784,Z 165.12,A -85,B 0,C 180,E1 -3090.204,E2 -3090.204} C_VEL
LIN {X 0,Y 558.767,Z 165.387,A -85,B 0,C 180,E1 -3090.433,E2 -3090.433} C_VEL
LIN {X 0,Y 558.055,Z 165.764,A -85,B 0,C 180,E1 -3090.705,E2 -3090.705} C_VEL
LIN {X 0,Y 552.372,Z 167.149,A -85,B 0,C 180,E1 -3091.49,E2 -3091.49} C_VEL
LIN {X 0,Y 551.673,Z 167.529,A -85,B 0,C 180,E1 -3091.767,E2 -3091.767} C_VEL
LIN {X 0,Y 551.692,Z 167.921,A -85,B 0,C 180,E1 -3092.103,E2 -3092.103} C_VEL
LIN {X 0,Y 553.038,Z 176.468,A -85,B 0,C 180,E1 -3092.34,E2 -3092.34} C_VEL
LIN {X 0,Y 552.879,Z 189.41,A -85,B 0,C 180,E1 -3092.766,E2 -3092.766} C_VEL
LIN {X 0,Y 552.644,Z 201.369,A -85,B 0,C 180,E1 -3093.313,E2 -3093.313} C_VEL
LIN {X 0,Y 552.445,Z 213.502,A -85,B 0,C 180,E1 -3094.038,E2 -3094.038} C_VEL
LIN {X 0,Y 552.315,Z 223.982,A -85,B 0,C 180,E1 -3094.834,E2 -3094.834} C_VEL
LIN {X 0,Y 552.158,Z 234.608,A -85,B 0,C 180,E1 -3095.838,E2 -3095.838} C_VEL
LIN {X 0,Y 551.988,Z 242.525,A -85,B 0,C 180,E1 -3096.756,E2 -3096.756} C_VEL
LIN {X 0,Y 551.871,Z 250.273,A -85,B 0,C 180,E1 -3097.855,E2 -3097.855} C_VEL
LIN {X 0,Y 551.8,Z 256.804,A -85,B 0,C 180,E1 -3099.02,E2 -3099.02} C_VEL
LIN {X 0,Y 551.742,Z 261.834,A -85,B 0,C 180,E1 -3100.157,E2 -3100.157} C_VEL
LIN {X 0,Y 551.731,Z 266.215,A -85,B 0,C 180,E1 -3101.481,E2 -3101.481} C_VEL
LIN {X 0,Y 551.695,Z 268.495,A -85,B 0,C 180,E1 -3102.466,E2 -3102.466} C_VEL
LIN {X 0,Y 551.669,Z 270.054,A -85,B 0,C 180,E1 -3103.466,E2 -3103.466} C_VEL
LIN {X 0,Y 551.669,Z 270.883,A -85,B 0,C 180,E1 -3104.486,E2 -3104.486} C_VEL
LIN {X 0,Y 551.669,Z 270.903,A -85,B 0,C 180,E1 -3105.519,E2 -3105.519} C_VEL
LIN {X 0,Y 551.668,Z 270.117,A -85,B 0,C 180,E1 -3106.564,E2 -3106.564} C_VEL
LIN {X 0,Y 551.696,Z 268.473,A -85,B 0,C 180,E1 -3107.633,E2 -3107.633} C_VEL
LIN {X 0,Y 551.729,Z 265.878,A -85,B 0,C 180,E1 -3108.724,E2 -3108.724} C_VEL
LIN {X 0,Y 551.741,Z 262.189,A -85,B 0,C 180,E1 -3109.841,E2 -3109.841} C_VEL
LIN {X 0,Y 551.831,Z 256.239,A -85,B 0,C 180,E1 -3111.185,E2 -3111.185} C_VEL
LIN {X 0,Y 551.885,Z 249.744,A -85,B 0,C 180,E1 -3112.319,E2 -3112.319} C_VEL
LIN {X 0,Y 551.996,Z 242.547,A -85,B 0,C 180,E1 -3113.332,E2 -3113.332} C_VEL
LIN {X 0,Y 552.173,Z 233.366,A -85,B 0,C 180,E1 -3114.381,E2 -3114.381} C_VEL
LIN {X 0,Y 552.306,Z 223.916,A -85,B 0,C 180,E1 -3115.262,E2 -3115.262} C_VEL
LIN {X 0,Y 552.469,Z 213.177,A -85,B 0,C 180,E1 -3116.073,E2 -3116.073} C_VEL
LIN {X 0,Y 552.641,Z 201.023,A -85,B 0,C 180,E1 -3116.795,E2 -3116.795} C_VEL
LIN {X 0,Y 552.889,Z 189.689,A -85,B 0,C 180,E1 -3117.312,E2 -3117.312} C_VEL
LIN {X 0,Y 553.039,Z 177.652,A -85,B 0,C 180,E1 -3117.718,E2 -3117.718} C_VEL
LIN {X 0,Y 552.467,Z 172.458,A -85,B 0,C 180,E1 -3117.866,E2 -3117.866} C_VEL
LIN {X 0,Y 551.686,Z 167.82,A -85,B 0,C 180,E1 -3118.003,E2 -3118.003} C_VEL
LIN {X 0,Y 551.718,Z 164.192,A -85,B 0,C 180,E1 -3121.049,E2 -3121.049} C_VEL
LIN {X 0,Y 551.749,Z 161.325,A -85,B 0,C 180,E1 -3123.524,E2 -3123.524} C_VEL
LIN {X 0,Y 551.753,Z 157.924,A -85,B 0,C 180,E1 -3126.505,E2 -3126.505} C_VEL
LIN {X 0,Y 551.771,Z 154.919,A -85,B 0,C 180,E1 -3129.106,E2 -3129.106} C_VEL
LIN {X 0,Y 551.794,Z 152.18,A -85,B 0,C 180,E1 -3131.433,E2 -3131.433} C_VEL
LIN {X 0,Y 551.837,Z 149.52,A -85,B 0,C 180,E1 -3133.729,E2 -3133.729} C_VEL
LIN {X 0,Y 551.897,Z 146.876,A -85,B 0,C 180,E1 -3135.998,E2 -3135.998} C_VEL
LIN {X 0,Y 551.979,Z 143.781,A -85,B 0,C 180,E1 -3138.632,E2 -3138.632} C_VEL
LIN {X 0,Y 552.142,Z 143.709,A -85,B 0,C 180,E1 -3141.214,E2 -3141.214} C_VEL
LIN {X 0,Y 552.197,Z 143.703,A -85,B 0,C 180,E1 -3144.156,E2 -3144.156} C_VEL
LIN {X 0,Y 552.202,Z 143.701,A -85,B 0,C 180,E1 -3147.082,E2 -3147.082} C_VEL
LIN {X 0,Y 552.23,Z 143.701,A -85,B 0,C 180,E1 -3150,E2 -3150} C_VEL
LIN {X 0,Y 552.201,Z 143.7,A -85,B 0,C 180,E1 -3152.918,E2 -3152.918} C_VEL
LIN {X 0,Y 552.196,Z 143.704,A -85,B 0,C 180,E1 -3155.844,E2 -3155.844} C_VEL
LIN {X 0,Y 552.155,Z 143.707,A -85,B 0,C 180,E1 -3158.786,E2 -3158.786} C_VEL
LIN {X 0,Y 552.16,Z 143.708,A -85,B 0,C 180,E1 -3161.75,E2 -3161.75} C_VEL
LIN {X 0,Y 552.133,Z 143.711,A -85,B 0,C 180,E1 -3164.748,E2 -3164.748} C_VEL
LIN {X 0,Y 552.11,Z 143.714,A -85,B 0,C 180,E1 -3167.788,E2 -3167.788} C_VEL
LIN {X 0,Y 552.128,Z 143.711,A -85,B 0,C 180,E1 -3170.101,E2 -3170.101} C_VEL
LIN {X 0,Y 552.093,Z 143.715,A -85,B 0,C 180,E1 -3172.451,E2 -3172.451} C_VEL
LIN {X 0,Y 552.153,Z 143.711,A -85,B 0,C 180,E1 -3175.351,E2 -3175.351} C_VEL
LIN {X 0,Y 552.117,Z 143.712,A -85,B 0,C 180,E1 -3178.098,E2 -3178.098} C_VEL
LIN {X 0,Y 552.103,Z 143.714,A -85,B 0,C 180,E1 -3180.609,E2 -3180.609} C_VEL
LIN {X 0,Y 552.12,Z 143.712,A -85,B 0,C 180,E1 -3183.186,E2 -3183.186} C_VEL
LIN {X 0,Y 552.083,Z 143.717,A -85,B 0,C 180,E1 -3185.844,E2 -3185.844} C_VEL
LIN {X 0,Y 552.123,Z 143.711,A -85,B 0,C 180,E1 -3189.062,E2 -3189.062} C_VEL
LIN {X 0,Y 552.135,Z 143.71,A -85,B 0,C 180,E1 -3191.445,E2 -3191.445} C_VEL
LIN {X 0,Y 552.093,Z 143.716,A -85,B 0,C 180,E1 -3194.532,E2 -3194.532} C_VEL
LIN {X 0,Y 552.127,Z 143.71,A -85,B 0,C 180,E1 -3197.585,E2 -3197.585} C_VEL
LIN {X 0,Y 552.129,Z 143.711,A -85,B 0,C 180,E1 -3200.473,E2 -3200.473} C_VEL
LIN {X 0,Y 552.109,Z 143.714,A -85,B 0,C 180,E1 -3203.317,E2 -3203.317} C_VEL
LIN {X 0,Y 552.105,Z 143.713,A -85,B 0,C 180,E1 -3205.938,E2 -3205.938} C_VEL
LIN {X 0,Y 552.118,Z 143.712,A -85,B 0,C 180,E1 -3208.541,E2 -3208.541} C_VEL
LIN {X 0,Y 552.124,Z 143.714,A -85,B 0,C 180,E1 -3211.438,E2 -3211.438} C_VEL
LIN {X 0,Y 552.13,Z 143.711,A -85,B 0,C 180,E1 -3214.356,E2 -3214.356} C_VEL
LIN {X 0,Y 552.098,Z 143.715,A -85,B 0,C 180,E1 -3216.758,E2 -3216.758} C_VEL
LIN {X 0,Y 552.121,Z 143.711,A -85,B 0,C 180,E1 -3219.12,E2 -3219.12} C_VEL
LIN {X 0,Y 552.12,Z 143.712,A -85,B 0,C 180,E1 -3221.445,E2 -3221.445} C_VEL
LIN {X 0,Y 552.115,Z 143.715,A -85,B 0,C 180,E1 -3223.738,E2 -3223.738} C_VEL
LIN {X 0,Y 552.132,Z 143.713,A -85,B 0,C 180,E1 -3226.005,E2 -3226.005} C_VEL
LIN {X 0,Y 552.164,Z 143.706,A -85,B 0,C 180,E1 -3228.994,E2 -3228.994} C_VEL
LIN {X 0,Y 552.149,Z 143.71,A -85,B 0,C 180,E1 -3231.952,E2 -3231.952} C_VEL
LIN {X 0,Y 552.226,Z 143.698,A -85,B 0,C 180,E1 -3234.889,E2 -3234.889} C_VEL
LIN {X 0,Y 552.227,Z 143.699,A -85,B 0,C 180,E1 -3237.812,E2 -3237.812} C_VEL
LIN {X 0,Y 552.243,Z 143.697,A -85,B 0,C 180,E1 -3240.73,E2 -3240.73} C_VEL
LIN {X 0,Y 552.205,Z 143.703,A -85,B 0,C 180,E1 -3242.918,E2 -3242.918} C_VEL
LIN {X 0,Y 552.201,Z 143.702,A -85,B 0,C 180,E1 -3245.844,E2 -3245.844} C_VEL
LIN {X 0,Y 552.144,Z 143.71,A -85,B 0,C 180,E1 -3248.786,E2 -3248.786} C_VEL
LIN {X 0,Y 552.166,Z 143.706,A -85,B 0,C 180,E1 -3251.751,E2 -3251.751} C_VEL
LIN {X 0,Y 552.131,Z 143.711,A -85,B 0,C 180,E1 -3254.749,E2 -3254.749} C_VEL
LIN {X 0,Y 552.111,Z 143.713,A -85,B 0,C 180,E1 -3257.789,E2 -3257.789} C_VEL
LIN {X 0,Y 552.129,Z 143.711,A -85,B 0,C 180,E1 -3260.102,E2 -3260.102} C_VEL
LIN {X 0,Y 552.094,Z 143.716,A -85,B 0,C 180,E1 -3262.451,E2 -3262.451} C_VEL
LIN {X 0,Y 552.159,Z 143.707,A -85,B 0,C 180,E1 -3265.351,E2 -3265.351} C_VEL
LIN {X 0,Y 552.113,Z 143.714,A -85,B 0,C 180,E1 -3268.099,E2 -3268.099} C_VEL
LIN {X 0,Y 552.104,Z 143.715,A -85,B 0,C 180,E1 -3270.61,E2 -3270.61} C_VEL
LIN {X 0,Y 552.108,Z 143.716,A -85,B 0,C 180,E1 -3273.187,E2 -3273.187} C_VEL
LIN {X 0,Y 552.088,Z 143.716,A -85,B 0,C 180,E1 -3275.844,E2 -3275.844} C_VEL
LIN {X 0,Y 552.118,Z 143.711,A -85,B 0,C 180,E1 -3278.589,E2 -3278.589} C_VEL
LIN {X 0,Y 552.123,Z 143.714,A -85,B 0,C 180,E1 -3281.446,E2 -3281.446} C_VEL
LIN {X 0,Y 552.096,Z 143.713,A -85,B 0,C 180,E1 -3284.532,E2 -3284.532} C_VEL
LIN {X 0,Y 552.132,Z 143.711,A -85,B 0,C 180,E1 -3287.585,E2 -3287.585} C_VEL
LIN {X 0,Y 552.135,Z 143.711,A -85,B 0,C 180,E1 -3290.473,E2 -3290.473} C_VEL
LIN {X 0,Y 552.133,Z 143.816,A -85,B 0,C 180,E1 -3292.512,E2 -3292.512} C_VEL
LIN {X 0,Y 552.913,Z 149.241,A -85,B 0,C 180,E1 -3294.439,E2 -3294.439} C_VEL
LIN {X 0,Y 552.827,Z 157.049,A -85,B 0,C 180,E1 -3297.04,E2 -3297.04} C_VEL
LIN {X 0,Y 552.66,Z 165.793,A -85,B 0,C 180,E1 -3299.853,E2 -3299.853} C_VEL
LIN {X 0,Y 552.489,Z 175.043,A -85,B 0,C 180,E1 -3302.746,E2 -3302.746} C_VEL
LIN {X 0,Y 552.352,Z 184.31,A -85,B 0,C 180,E1 -3305.574,E2 -3305.574} C_VEL
LIN {X 0,Y 552.212,Z 193.577,A -85,B 0,C 180,E1 -3308.341,E2 -3308.341} C_VEL
LIN {X 0,Y 552.085,Z 202.844,A -85,B 0,C 180,E1 -3311.058,E2 -3311.058} C_VEL
LIN {X 0,Y 551.992,Z 213.436,A -85,B 0,C 180,E1 -3314.113,E2 -3314.113} C_VEL
LIN {X 0,Y 551.889,Z 223.53,A -85,B 0,C 180,E1 -3316.983,E2 -3316.983} C_VEL
LIN {X 0,Y 553.099,Z 232.526,A -85,B 0,C 180,E1 -3317.199,E2 -3317.199} C_VEL
LIN {X 0,Y 552.962,Z 245.18,A -85,B 0,C 180,E1 -3317.569,E2 -3317.569} C_VEL
LIN {X 0,Y 552.744,Z 257.487,A -85,B 0,C 180,E1 -3318.076,E2 -3318.076} C_VEL
LIN {X 0,Y 552.576,Z 269.235,A -85,B 0,C 180,E1 -3318.718,E2 -3318.718} C_VEL
LIN {X 0,Y 552.43,Z 279.928,A -85,B 0,C 180,E1 -3319.463,E2 -3319.463} C_VEL
LIN {X 0,Y 552.233,Z 289.602,A -85,B 0,C 180,E1 -3320.292,E2 -3320.292} C_VEL
LIN {X 0,Y 552.079,Z 298.414,A -85,B 0,C 180,E1 -3321.213,E2 -3321.213} C_VEL
LIN {X 0,Y 551.95,Z 307.001,A -85,B 0,C 180,E1 -3322.317,E2 -3322.317} C_VEL
LIN {X 0,Y 551.823,Z 313.868,A -85,B 0,C 180,E1 -3323.418,E2 -3323.418} C_VEL
LIN {X 0,Y 551.804,Z 319.366,A -85,B 0,C 180,E1 -3324.519,E2 -3324.519} C_VEL
LIN {X 0,Y 551.764,Z 323.678,A -85,B 0,C 180,E1 -3325.617,E2 -3325.617} C_VEL
LIN {X 0,Y 551.75,Z 325.957,A -85,B 0,C 180,E1 -3326.349,E2 -3326.349} C_VEL
LIN {X 0,Y 551.724,Z 327.809,A -85,B 0,C 180,E1 -3327.079,E2 -3327.079} C_VEL
LIN {X 0,Y 551.645,Z 330.185,A -85,B 0,C 180,E1 -3328.54,E2 -3328.54} C_VEL
LIN {X 0,Y 551.64,Z 331,A -85,B 0,C 180,E1 -3330,E2 -3330} C_VEL
LIN {X 0,Y 551.645,Z 330.186,A -85,B 0,C 180,E1 -3331.46,E2 -3331.46} C_VEL
LIN {X 0,Y 551.657,Z 329.2,A -85,B 0,C 180,E1 -3332.19,E2 -3332.19} C_VEL
LIN {X 0,Y 551.724,Z 327.809,A -85,B 0,C 180,E1 -3332.921,E2 -3332.921} C_VEL
LIN {X 0,Y 551.764,Z 324.895,A -85,B 0,C 180,E1 -3334.017,E2 -3334.017} C_VEL
LIN {X 0,Y 551.724,Z 320.949,A -85,B 0,C 180,E1 -3335.116,E2 -3335.116} C_VEL
LIN {X 0,Y 551.823,Z 315.203,A -85,B 0,C 180,E1 -3336.339,E2 -3336.339} C_VEL
LIN {X 0,Y 551.927,Z 308.236,A -85,B 0,C 180,E1 -3337.5,E2 -3337.5} C_VEL
LIN {X 0,Y 552.082,Z 299.989,A -85,B 0,C 180,E1 -3338.603,E2 -3338.603} C_VEL
LIN {X 0,Y 552.201,Z 291.536,A -85,B 0,C 180,E1 -3339.524,E2 -3339.524} C_VEL
LIN {X 0,Y 552.423,Z 281.094,A -85,B 0,C 180,E1 -3340.445,E2 -3340.445} C_VEL
LIN {X 0,Y 552.579,Z 269.348,A -85,B 0,C 180,E1 -3341.275,E2 -3341.275} C_VEL
LIN {X 0,Y 552.742,Z 257.48,A -85,B 0,C 180,E1 -3341.924,E2 -3341.924} C_VEL
LIN {X 0,Y 552.927,Z 245.168,A -85,B 0,C 180,E1 -3342.432,E2 -3342.432} C_VEL
LIN {X 0,Y 553.079,Z 232.513,A -85,B 0,C 180,E1 -3342.802,E2 -3342.802} C_VEL
LIN {X 0,Y 552.355,Z 226.498,A -85,B 0,C 180,E1 -3342.944,E2 -3342.944} C_VEL
LIN {X 0,Y 551.889,Z 223.53,A -85,B 0,C 180,E1 -3343.017,E2 -3343.017} C_VEL
LIN {X 0,Y 551.992,Z 213.435,A -85,B 0,C 180,E1 -3345.887,E2 -3345.887} C_VEL
LIN {X 0,Y 552.086,Z 202.844,A -85,B 0,C 180,E1 -3348.942,E2 -3348.942} C_VEL
LIN {X 0,Y 552.255,Z 192.254,A -85,B 0,C 180,E1 -3352.05,E2 -3352.05} C_VEL
LIN {X 0,Y 552.37,Z 182.985,A -85,B 0,C 180,E1 -3354.827,E2 -3354.827} C_VEL
LIN {X 0,Y 552.529,Z 173.718,A -85,B 0,C 180,E1 -3357.663,E2 -3357.663} C_VEL
LIN {X 0,Y 552.676,Z 164.45,A -85,B 0,C 180,E1 -3360.574,E2 -3360.574} C_VEL
LIN {X 0,Y 552.896,Z 155.183,A -85,B 0,C 180,E1 -3363.569,E2 -3363.569} C_VEL
LIN {X 0,Y 552.874,Z 148.439,A -85,B 0,C 180,E1 -3365.785,E2 -3365.785} C_VEL
LIN {X 0,Y 552.116,Z 143.715,A -85,B 0,C 180,E1 -3367.547,E2 -3367.547} C_VEL
LIN {X 0,Y 552.114,Z 143.715,A -85,B 0,C 180,E1 -3370.481,E2 -3370.481} C_VEL
LIN {X 0,Y 552.124,Z 143.713,A -85,B 0,C 180,E1 -3373.485,E2 -3373.485} C_VEL
LIN {X 0,Y 552.111,Z 143.715,A -85,B 0,C 180,E1 -3376.576,E2 -3376.576} C_VEL
LIN {X 0,Y 552.124,Z 143.714,A -85,B 0,C 180,E1 -3379.52,E2 -3379.52} C_VEL
LIN {X 0,Y 552.097,Z 143.718,A -85,B 0,C 180,E1 -3382.336,E2 -3382.336} C_VEL
LIN {X 0,Y 552.092,Z 143.717,A -85,B 0,C 180,E1 -3385.051,E2 -3385.051} C_VEL
LIN {X 0,Y 552.131,Z 143.711,A -85,B 0,C 180,E1 -3387.682,E2 -3387.682} C_VEL
LIN {X 0,Y 552.117,Z 143.714,A -85,B 0,C 180,E1 -3390.235,E2 -3390.235} C_VEL
LIN {X 0,Y 552.144,Z 143.709,A -85,B 0,C 180,E1 -3393,E2 -3393} C_VEL
LIN {X 0,Y 552.118,Z 143.713,A -85,B 0,C 180,E1 -3395.161,E2 -3395.161} C_VEL
LIN {X 0,Y 552.131,Z 143.712,A -85,B 0,C 180,E1 -3398.337,E2 -3398.337} C_VEL
LIN {X 0,Y 552.156,Z 143.709,A -85,B 0,C 180,E1 -3400.674,E2 -3400.674} C_VEL
LIN {X 0,Y 552.118,Z 143.713,A -85,B 0,C 180,E1 -3403.737,E2 -3403.737} C_VEL
LIN {X 0,Y 552.141,Z 143.71,A -85,B 0,C 180,E1 -3406.004,E2 -3406.004} C_VEL
LIN {X 0,Y 552.168,Z 143.707,A -85,B 0,C 180,E1 -3408.993,E2 -3408.993} C_VEL
LIN {X 0,Y 552.163,Z 143.707,A -85,B 0,C 180,E1 -3411.951,E2 -3411.951} C_VEL
LIN {X 0,Y 552.232,Z 143.699,A -85,B 0,C 180,E1 -3414.889,E2 -3414.889} C_VEL
LIN {X 0,Y 552.23,Z 143.7,A -85,B 0,C 180,E1 -3417.812,E2 -3417.812} C_VEL
LIN {X 0,Y 552.248,Z 143.698,A -85,B 0,C 180,E1 -3420.729,E2 -3420.729} C_VEL
LIN {X 0,Y 552.208,Z 143.702,A -85,B 0,C 180,E1 -3422.918,E2 -3422.918} C_VEL
LIN {X 0,Y 552.2,Z 143.705,A -85,B 0,C 180,E1 -3425.843,E2 -3425.843} C_VEL
LIN {X 0,Y 552.146,Z 143.712,A -85,B 0,C 180,E1 -3428.785,E2 -3428.785} C_VEL
LIN {X 0,Y 551.968,Z 143.834,A -85,B 0,C 180,E1 -3431.01,E2 -3431.01} C_VEL
LIN {X 0,Y 551.947,Z 147.34,A -85,B 0,C 180,E1 -3434,E2 -3434} C_VEL
LIN {X 0,Y 551.91,Z 151.082,A -85,B 0,C 180,E1 -3437.244,E2 -3437.244} C_VEL
LIN {X 0,Y 551.791,Z 154.355,A -85,B 0,C 180,E1 -3440.114,E2 -3440.114} C_VEL
LIN {X 0,Y 551.754,Z 156.967,A -85,B 0,C 180,E1 -3442.465,E2 -3442.465} C_VEL
LIN {X 0,Y 551.768,Z 160.223,A -85,B 0,C 180,E1 -3445.264,E2 -3445.264} C_VEL
LIN {X 0,Y 551.755,Z 163.349,A -85,B 0,C 180,E1 -3448.118,E2 -3448.118} C_VEL
LIN {X 0,Y 551.685,Z 166.213,A -85,B 0,C 180,E1 -3450.634,E2 -3450.634} C_VEL
LIN {X 0,Y 551.673,Z 167.529,A -85,B 0,C 180,E1 -3451.767,E2 -3451.767} C_VEL
LIN {X 0,Y 551.659,Z 168.635,A -85,B 0,C 180,E1 -3451.975,E2 -3451.975} C_VEL
LIN {X 0,Y 551.589,Z 171.614,A -85,B 0,C 180,E1 -3452.159,E2 -3452.159} C_VEL
LIN {X 0,Y 550.757,Z 181.351,A -85,B 0,C 180,E1 -3452.426,E2 -3452.426} C_VEL
LIN {X 0,Y 546.611,Z 193.134,A -85,B 0,C 180,E1 -3452.752,E2 -3452.752} C_VEL
LIN {X 0,Y 545.844,Z 196.718,A -85,B 0,C 180,E1 -3452.911,E2 -3452.911} C_VEL
LIN {X 0,Y 545.584,Z 208.862,A -85,B 0,C 180,E1 -3453.568,E2 -3453.568} C_VEL
LIN {X 0,Y 545.415,Z 220.275,A -85,B 0,C 180,E1 -3454.372,E2 -3454.372} C_VEL
LIN {X 0,Y 545.209,Z 231.235,A -85,B 0,C 180,E1 -3455.342,E2 -3455.342} C_VEL
LIN {X 0,Y 545.007,Z 240.614,A -85,B 0,C 180,E1 -3456.383,E2 -3456.383} C_VEL
LIN {X 0,Y 544.86,Z 248.794,A -85,B 0,C 180,E1 -3457.513,E2 -3457.513} C_VEL
LIN {X 0,Y 544.753,Z 255.845,A -85,B 0,C 180,E1 -3458.734,E2 -3458.734} C_VEL
LIN {X 0,Y 544.695,Z 260.269,A -85,B 0,C 180,E1 -3459.699,E2 -3459.699} C_VEL
LIN {X 0,Y 544.627,Z 264.2,A -85,B 0,C 180,E1 -3460.761,E2 -3460.761} C_VEL
LIN {X 0,Y 544.64,Z 267.929,A -85,B 0,C 180,E1 -3462.144,E2 -3462.144} C_VEL
LIN {X 0,Y 544.576,Z 269.695,A -85,B 0,C 180,E1 -3463.155,E2 -3463.155} C_VEL
LIN {X 0,Y 544.559,Z 270.704,A -85,B 0,C 180,E1 -3464.179,E2 -3464.179} C_VEL
LIN {X 0,Y 544.557,Z 270.969,A -85,B 0,C 180,E1 -3465.22,E2 -3465.22} C_VEL
LIN {X 0,Y 544.567,Z 270.446,A -85,B 0,C 180,E1 -3466.279,E2 -3466.279} C_VEL
LIN {X 0,Y 544.589,Z 269.052,A -85,B 0,C 180,E1 -3467.357,E2 -3467.357} C_VEL
LIN {X 0,Y 544.626,Z 265.674,A -85,B 0,C 180,E1 -3468.843,E2 -3468.843} C_VEL
LIN {X 0,Y 544.664,Z 262.506,A -85,B 0,C 180,E1 -3469.821,E2 -3469.821} C_VEL
LIN {X 0,Y 544.713,Z 257.445,A -85,B 0,C 180,E1 -3471.025,E2 -3471.025} C_VEL
LIN {X 0,Y 544.803,Z 250.631,A -85,B 0,C 180,E1 -3472.286,E2 -3472.286} C_VEL
LIN {X 0,Y 544.964,Z 243.355,A -85,B 0,C 180,E1 -3473.357,E2 -3473.357} C_VEL
LIN {X 0,Y 545.133,Z 234.783,A -85,B 0,C 180,E1 -3474.377,E2 -3474.377} C_VEL
LIN {X 0,Y 545.309,Z 224.809,A -85,B 0,C 180,E1 -3475.341,E2 -3475.341} C_VEL
LIN {X 0,Y 545.477,Z 214.675,A -85,B 0,C 180,E1 -3476.135,E2 -3476.135} C_VEL
LIN {X 0,Y 545.637,Z 203.232,A -85,B 0,C 180,E1 -3476.847,E2 -3476.847} C_VEL
LIN {X 0,Y 545.956,Z 190.824,A -85,B 0,C 180,E1 -3477.435,E2 -3477.435} C_VEL
LIN {X 0,Y 546.118,Z 177.892,A -85,B 0,C 180,E1 -3477.883,E2 -3477.883} C_VEL
LIN {X 0,Y 544.592,Z 168.228,A -85,B 0,C 180,E1 -3478.157,E2 -3478.157} C_VEL
LIN {X 0,Y 544.615,Z 165.276,A -85,B 0,C 180,E1 -3480.635,E2 -3480.635} C_VEL
LIN {X 0,Y 544.689,Z 162.368,A -85,B 0,C 180,E1 -3483.154,E2 -3483.154} C_VEL
LIN {X 0,Y 544.665,Z 159.562,A -85,B 0,C 180,E1 -3485.612,E2 -3485.612} C_VEL
LIN {X 0,Y 544.69,Z 155.853,A -85,B 0,C 180,E1 -3488.821,E2 -3488.821} C_VEL
LIN {X 0,Y 544.717,Z 153.092,A -85,B 0,C 180,E1 -3491.182,E2 -3491.182} C_VEL
LIN {X 0,Y 544.783,Z 150.391,A -85,B 0,C 180,E1 -3493.512,E2 -3493.512} C_VEL
LIN {X 0,Y 544.822,Z 147.72,A -85,B 0,C 180,E1 -3495.813,E2 -3495.813} C_VEL
LIN {X 0,Y 544.912,Z 144.613,A -85,B 0,C 180,E1 -3498.58,E2 -3498.58} C_VEL
LIN {X 0,Y 545.096,Z 144.586,A -85,B 0,C 180,E1 -3501.099,E2 -3501.099} C_VEL
LIN {X 0,Y 545.167,Z 144.58,A -85,B 0,C 180,E1 -3504.08,E2 -3504.08} C_VEL
LIN {X 0,Y 545.169,Z 144.577,A -85,B 0,C 180,E1 -3507.044,E2 -3507.044} C_VEL
LIN {X 0,Y 545.2,Z 144.577,A -85,B 0,C 180,E1 -3510,E2 -3510} C_VEL
LIN {X 0,Y 545.168,Z 144.576,A -85,B 0,C 180,E1 -3512.956,E2 -3512.956} C_VEL
LIN {X 0,Y 545.166,Z 144.58,A -85,B 0,C 180,E1 -3515.919,E2 -3515.919} C_VEL
LIN {X 0,Y 545.114,Z 144.584,A -85,B 0,C 180,E1 -3518.9,E2 -3518.9} C_VEL
LIN {X 0,Y 545.132,Z 144.584,A -85,B 0,C 180,E1 -3521.904,E2 -3521.904} C_VEL
LIN {X 0,Y 545.082,Z 144.588,A -85,B 0,C 180,E1 -3524.944,E2 -3524.944} C_VEL
LIN {X 0,Y 545.078,Z 144.592,A -85,B 0,C 180,E1 -3528.026,E2 -3528.026} C_VEL
LIN {X 0,Y 545.092,Z 144.589,A -85,B 0,C 180,E1 -3530.372,E2 -3530.372} C_VEL
LIN {X 0,Y 545.09,Z 144.588,A -85,B 0,C 180,E1 -3533.559,E2 -3533.559} C_VEL
LIN {X 0,Y 545.077,Z 144.589,A -85,B 0,C 180,E1 -3536.001,E2 -3536.001} C_VEL
LIN {X 0,Y 545.087,Z 144.588,A -85,B 0,C 180,E1 -3538.749,E2 -3538.749} C_VEL
LIN {X 0,Y 545.056,Z 144.592,A -85,B 0,C 180,E1 -3541.679,E2 -3541.679} C_VEL
LIN {X 0,Y 545.073,Z 144.588,A -85,B 0,C 180,E1 -3544.392,E2 -3544.392} C_VEL
LIN {X 0,Y 545.034,Z 144.597,A -85,B 0,C 180,E1 -3547.304,E2 -3547.304} C_VEL
LIN {X 0,Y 545.07,Z 144.59,A -85,B 0,C 180,E1 -3550.142,E2 -3550.142} C_VEL
LIN {X 0,Y 545.076,Z 144.59,A -85,B 0,C 180,E1 -3553.107,E2 -3553.107} C_VEL
LIN {X 0,Y 545.065,Z 144.591,A -85,B 0,C 180,E1 -3556.225,E2 -3556.225} C_VEL
LIN {X 0,Y 545.08,Z 144.589,A -85,B 0,C 180,E1 -3558.886,E2 -3558.886} C_VEL
LIN {X 0,Y 545.08,Z 144.591,A -85,B 0,C 180,E1 -3560.819,E2 -3560.819} C_VEL
LIN {X 0,Y 545.048,Z 144.592,A -85,B 0,C 180,E1 -3563.621,E2 -3563.621} C_VEL
LIN {X 0,Y 545.051,Z 144.592,A -85,B 0,C 180,E1 -3566.328,E2 -3566.328} C_VEL
LIN {X 0,Y 545.066,Z 144.592,A -85,B 0,C 180,E1 -3568.953,E2 -3568.953} C_VEL
LIN {X 0,Y 545.101,Z 144.588,A -85,B 0,C 180,E1 -3571.508,E2 -3571.508} C_VEL
LIN {X 0,Y 545.095,Z 144.587,A -85,B 0,C 180,E1 -3574.492,E2 -3574.492} C_VEL
LIN {X 0,Y 545.038,Z 144.594,A -85,B 0,C 180,E1 -3577.243,E2 -3577.243} C_VEL
LIN {X 0,Y 545.121,Z 144.584,A -85,B 0,C 180,E1 -3580.415,E2 -3580.415} C_VEL
LIN {X 0,Y 545.066,Z 144.592,A -85,B 0,C 180,E1 -3583.521,E2 -3583.521} C_VEL
LIN {X 0,Y 545.092,Z 144.588,A -85,B 0,C 180,E1 -3585.82,E2 -3585.82} C_VEL
LIN {X 0,Y 545.119,Z 144.583,A -85,B 0,C 180,E1 -3588.85,E2 -3588.85} C_VEL
LIN {X 0,Y 545.098,Z 144.587,A -85,B 0,C 180,E1 -3591.847,E2 -3591.847} C_VEL
LIN {X 0,Y 545.203,Z 144.573,A -85,B 0,C 180,E1 -3594.823,E2 -3594.823} C_VEL
LIN {X 0,Y 545.198,Z 144.574,A -85,B 0,C 180,E1 -3597.784,E2 -3597.784} C_VEL
LIN {X 0,Y 545.214,Z 144.572,A -85,B 0,C 180,E1 -3600.739,E2 -3600.739} C_VEL
LIN {X 0,Y 545.172,Z 144.579,A -85,B 0,C 180,E1 -3602.956,E2 -3602.956} C_VEL
LIN {X 0,Y 545.171,Z 144.577,A -85,B 0,C 180,E1 -3605.92,E2 -3605.92} C_VEL
LIN {X 0,Y 545.105,Z 144.587,A -85,B 0,C 180,E1 -3608.901,E2 -3608.901} C_VEL
LIN {X 0,Y 545.138,Z 144.581,A -85,B 0,C 180,E1 -3611.904,E2 -3611.904} C_VEL
LIN {X 0,Y 545.084,Z 144.59,A -85,B 0,C 180,E1 -3614.944,E2 -3614.944} C_VEL
LIN {X 0,Y 545.079,Z 144.589,A -85,B 0,C 180,E1 -3618.026,E2 -3618.026} C_VEL
LIN {X 0,Y 545.094,Z 144.586,A -85,B 0,C 180,E1 -3620.372,E2 -3620.372} C_VEL
LIN {X 0,Y 545.079,Z 144.591,A -85,B 0,C 180,E1 -3623.56,E2 -3623.56} C_VEL
LIN {X 0,Y 545.083,Z 144.589,A -85,B 0,C 180,E1 -3626.001,E2 -3626.001} C_VEL
LIN {X 0,Y 545.091,Z 144.587,A -85,B 0,C 180,E1 -3628.748,E2 -3628.748} C_VEL
LIN {X 0,Y 545.06,Z 144.593,A -85,B 0,C 180,E1 -3631.679,E2 -3631.679} C_VEL
LIN {X 0,Y 545.061,Z 144.592,A -85,B 0,C 180,E1 -3634.565,E2 -3634.565} C_VEL
LIN {X 0,Y 545.038,Z 144.594,A -85,B 0,C 180,E1 -3637.304,E2 -3637.304} C_VEL
LIN {X 0,Y 545.067,Z 144.591,A -85,B 0,C 180,E1 -3640.143,E2 -3640.143} C_VEL
LIN {X 0,Y 545.081,Z 144.587,A -85,B 0,C 180,E1 -3643.107,E2 -3643.107} C_VEL
LIN {X 0,Y 545.052,Z 144.592,A -85,B 0,C 180,E1 -3646.226,E2 -3646.226} C_VEL
LIN {X 0,Y 545.084,Z 144.59,A -85,B 0,C 180,E1 -3648.886,E2 -3648.886} C_VEL
LIN {X 0,Y 545.085,Z 144.59,A -85,B 0,C 180,E1 -3650.819,E2 -3650.819} C_VEL
LIN {X 0,Y 545.087,Z 144.659,A -85,B 0,C 180,E1 -3652.234,E2 -3652.234} C_VEL
LIN {X 0,Y 545.974,Z 150.051,A -85,B 0,C 180,E1 -3654.19,E2 -3654.19} C_VEL
LIN {X 0,Y 545.887,Z 157.782,A -85,B 0,C 180,E1 -3656.808,E2 -3656.808} C_VEL
LIN {X 0,Y 545.667,Z 167.099,A -85,B 0,C 180,E1 -3659.847,E2 -3659.847} C_VEL
LIN {X 0,Y 545.505,Z 176.24,A -85,B 0,C 180,E1 -3662.743,E2 -3662.743} C_VEL
LIN {X 0,Y 545.342,Z 185.634,A -85,B 0,C 180,E1 -3665.645,E2 -3665.645} C_VEL
LIN {X 0,Y 545.173,Z 195.064,A -85,B 0,C 180,E1 -3668.493,E2 -3668.493} C_VEL
LIN {X 0,Y 545.029,Z 204.168,A -85,B 0,C 180,E1 -3671.194,E2 -3671.194} C_VEL
LIN {X 0,Y 544.92,Z 214.76,A -85,B 0,C 180,E1 -3674.286,E2 -3674.286} C_VEL
LIN {X 0,Y 544.805,Z 223.53,A -85,B 0,C 180,E1 -3676.811,E2 -3676.811} C_VEL
LIN {X 0,Y 546.18,Z 233.441,A -85,B 0,C 180,E1 -3677.057,E2 -3677.057} C_VEL
LIN {X 0,Y 546.019,Z 245.179,A -85,B 0,C 180,E1 -3677.408,E2 -3677.408} C_VEL
LIN {X 0,Y 545.785,Z 257.488,A -85,B 0,C 180,E1 -3677.922,E2 -3677.922} C_VEL
LIN {X 0,Y 545.584,Z 269.618,A -85,B 0,C 180,E1 -3678.596,E2 -3678.596} C_VEL
LIN {X 0,Y 545.419,Z 281.099,A -85,B 0,C 180,E1 -3679.42,E2 -3679.42} C_VEL
LIN {X 0,Y 545.165,Z 291.539,A -85,B 0,C 180,E1 -3680.352,E2 -3680.352} C_VEL
LIN {X 0,Y 545.029,Z 299.991,A -85,B 0,C 180,E1 -3681.285,E2 -3681.285} C_VEL
LIN {X 0,Y 544.86,Z 308.238,A -85,B 0,C 180,E1 -3682.403,E2 -3682.403} C_VEL
LIN {X 0,Y 544.734,Z 315.617,A -85,B 0,C 180,E1 -3683.655,E2 -3683.655} C_VEL
LIN {X 0,Y 544.653,Z 320.95,A -85,B 0,C 180,E1 -3684.818,E2 -3684.818} C_VEL
LIN {X 0,Y 544.684,Z 324.896,A -85,B 0,C 180,E1 -3685.931,E2 -3685.931} C_VEL
LIN {X 0,Y 544.65,Z 327.809,A -85,B 0,C 180,E1 -3687.041,E2 -3687.041} C_VEL
LIN {X 0,Y 544.546,Z 330.186,A -85,B 0,C 180,E1 -3688.521,E2 -3688.521} C_VEL
LIN {X 0,Y 544.541,Z 331,A -85,B 0,C 180,E1 -3690,E2 -3690} C_VEL
LIN {X 0,Y 544.546,Z 330.186,A -85,B 0,C 180,E1 -3691.479,E2 -3691.479} C_VEL
LIN {X 0,Y 544.65,Z 327.81,A -85,B 0,C 180,E1 -3692.959,E2 -3692.959} C_VEL
LIN {X 0,Y 544.684,Z 324.895,A -85,B 0,C 180,E1 -3694.07,E2 -3694.07} C_VEL
LIN {X 0,Y 544.653,Z 320.948,A -85,B 0,C 180,E1 -3695.182,E2 -3695.182} C_VEL
LIN {X 0,Y 544.735,Z 315.611,A -85,B 0,C 180,E1 -3696.346,E2 -3696.346} C_VEL
LIN {X 0,Y 544.86,Z 308.236,A -85,B 0,C 180,E1 -3697.598,E2 -3697.598} C_VEL
LIN {X 0,Y 545.029,Z 299.989,A -85,B 0,C 180,E1 -3698.715,E2 -3698.715} C_VEL
LIN {X 0,Y 545.165,Z 291.536,A -85,B 0,C 180,E1 -3699.648,E2 -3699.648} C_VEL
LIN {X 0,Y 545.42,Z 281.095,A -85,B 0,C 180,E1 -3700.581,E2 -3700.581} C_VEL
LIN {X 0,Y 545.606,Z 269.662,A -85,B 0,C 180,E1 -3701.401,E2 -3701.401} C_VEL
LIN {X 0,Y 545.763,Z 259.408,A -85,B 0,C 180,E1 -3701.985,E2 -3701.985} C_VEL
LIN {X 0,Y 545.986,Z 247.758,A -85,B 0,C 180,E1 -3702.499,E2 -3702.499} C_VEL
LIN {X 0,Y 546.137,Z 234.342,A -85,B 0,C 180,E1 -3702.92,E2 -3702.92} C_VEL
LIN {X 0,Y 545.811,Z 229.726,A -85,B 0,C 180,E1 -3703.036,E2 -3703.036} C_VEL
LIN {X 0,Y 544.805,Z 223.53,A -85,B 0,C 180,E1 -3703.189,E2 -3703.189} C_VEL
LIN {X 0,Y 544.936,Z 213.435,A -85,B 0,C 180,E1 -3706.098,E2 -3706.098} C_VEL
LIN {X 0,Y 545.069,Z 202.844,A -85,B 0,C 180,E1 -3709.196,E2 -3709.196} C_VEL
LIN {X 0,Y 545.219,Z 192.252,A -85,B 0,C 180,E1 -3712.35,E2 -3712.35} C_VEL
LIN {X 0,Y 545.36,Z 182.985,A -85,B 0,C 180,E1 -3715.168,E2 -3715.168} C_VEL
LIN {X 0,Y 545.563,Z 173.718,A -85,B 0,C 180,E1 -3718.047,E2 -3718.047} C_VEL
LIN {X 0,Y 545.738,Z 164.45,A -85,B 0,C 180,E1 -3721.006,E2 -3721.006} C_VEL
LIN {X 0,Y 545.943,Z 155.1,A -85,B 0,C 180,E1 -3724.055,E2 -3724.055} C_VEL
LIN {X 0,Y 545.919,Z 149.86,A -85,B 0,C 180,E1 -3725.802,E2 -3725.802} C_VEL
LIN {X 0,Y 545.073,Z 144.593,A -85,B 0,C 180,E1 -3727.813,E2 -3727.813} C_VEL
LIN {X 0,Y 545.086,Z 144.59,A -85,B 0,C 180,E1 -3730.473,E2 -3730.473} C_VEL
LIN {X 0,Y 545.083,Z 144.589,A -85,B 0,C 180,E1 -3733.107,E2 -3733.107} C_VEL
LIN {X 0,Y 545.072,Z 144.593,A -85,B 0,C 180,E1 -3736.224,E2 -3736.224} C_VEL
LIN {X 0,Y 545.096,Z 144.589,A -85,B 0,C 180,E1 -3738.886,E2 -3738.886} C_VEL
LIN {X 0,Y 545.057,Z 144.593,A -85,B 0,C 180,E1 -3741.763,E2 -3741.763} C_VEL
LIN {X 0,Y 545.043,Z 144.595,A -85,B 0,C 180,E1 -3744.532,E2 -3744.532} C_VEL
LIN {X 0,Y 545.087,Z 144.59,A -85,B 0,C 180,E1 -3747.212,E2 -3747.212} C_VEL
LIN {X 0,Y 545.07,Z 144.591,A -85,B 0,C 180,E1 -3749.81,E2 -3749.81} C_VEL
LIN {X 0,Y 545.094,Z 144.59,A -85,B 0,C 180,E1 -3752.344,E2 -3752.344} C_VEL
LIN {X 0,Y 545.122,Z 144.584,A -85,B 0,C 180,E1 -3754.82,E2 -3754.82} C_VEL
LIN {X 0,Y 545.042,Z 144.595,A -85,B 0,C 180,E1 -3757.242,E2 -3757.242} C_VEL
LIN {X 0,Y 545.121,Z 144.586,A -85,B 0,C 180,E1 -3760.415,E2 -3760.415} C_VEL
LIN {X 0,Y 545.069,Z 144.593,A -85,B 0,C 180,E1 -3763.521,E2 -3763.521} C_VEL
LIN {X 0,Y 545.1,Z 144.587,A -85,B 0,C 180,E1 -3765.82,E2 -3765.82} C_VEL
LIN {X 0,Y 545.123,Z 144.585,A -85,B 0,C 180,E1 -3768.849,E2 -3768.849} C_VEL
LIN {X 0,Y 545.134,Z 144.583,A -85,B 0,C 180,E1 -3771.847,E2 -3771.847} C_VEL
LIN {X 0,Y 545.208,Z 144.574,A -85,B 0,C 180,E1 -3774.823,E2 -3774.823} C_VEL
LIN {X 0,Y 545.201,Z 144.576,A -85,B 0,C 180,E1 -3777.783,E2 -3777.783} C_VEL
LIN {X 0,Y 545.218,Z 144.574,A -85,B 0,C 180,E1 -3780.738,E2 -3780.738} C_VEL
LIN {X 0,Y 545.175,Z 144.578,A -85,B 0,C 180,E1 -3782.955,E2 -3782.955} C_VEL
LIN {X 0,Y 545.172,Z 144.58,A -85,B 0,C 180,E1 -3785.919,E2 -3785.919} C_VEL
LIN {X 0,Y 545.101,Z 144.588,A -85,B 0,C 180,E1 -3788.9,E2 -3788.9} C_VEL
LIN {X 0,Y 544.919,Z 144.754,A -85,B 0,C 180,E1 -3791.154,E2 -3791.154} C_VEL
LIN {X 0,Y 544.89,Z 148.851,A -85,B 0,C 180,E1 -3794.68,E2 -3794.68} C_VEL
LIN {X 0,Y 544.835,Z 151.889,A -85,B 0,C 180,E1 -3797.34,E2 -3797.34} C_VEL
LIN {X 0,Y 544.732,Z 155.318,A -85,B 0,C 180,E1 -3800.386,E2 -3800.386} C_VEL
LIN {X 0,Y 544.713,Z 158.909,A -85,B 0,C 180,E1 -3803.576,E2 -3803.576} C_VEL
LIN {X 0,Y 544.695,Z 161.694,A -85,B 0,C 180,E1 -3806.02,E2 -3806.02} C_VEL
LIN {X 0,Y 544.657,Z 164.601,A -85,B 0,C 180,E1 -3808.664,E2 -3808.664} C_VEL
LIN {X 0,Y 544.625,Z 168.261,A -85,B 0,C 180,E1 -3811.841,E2 -3811.841} C_VEL
LIN {X 0,Y 544.619,Z 168.397,A -85,B 0,C 180,E1 -3811.943,E2 -3811.943} C_VEL
LIN {X 0,Y 546.125,Z 177.574,A -85,B 0,C 180,E1 -3812.198,E2 -3812.198} C_VEL
LIN {X 0,Y 545.945,Z 190.042,A -85,B 0,C 180,E1 -3812.619,E2 -3812.619} C_VEL
LIN {X 0,Y 545.844,Z 196.718,A -85,B 0,C 180,E1 -3812.911,E2 -3812.911} C_VEL
LIN {X 0,Y 545.104,Z 202.106,A -85,B 0,C 180,E1 -3813.164,E2 -3813.164} C_VEL
LIN {X 0,Y 542.149,Z 210.632,A -85,B 0,C 180,E1 -3813.597,E2 -3813.597} C_VEL
LIN {X 0,Y 539.187,Z 218.773,A -85,B 0,C 180,E1 -3814.099,E2 -3814.099} C_VEL
LIN {X 0,Y 538.422,Z 223.494,A -85,B 0,C 180,E1 -3814.463,E2 -3814.463} C_VEL
LIN {X 0,Y 538.189,Z 233.558,A -85,B 0,C 180,E1 -3815.413,E2 -3815.413} C_VEL
LIN {X 0,Y 537.975,Z 242.594,A -85,B 0,C 180,E1 -3816.47,E2 -3816.47} C_VEL
LIN {X 0,Y 537.816,Z 249.703,A -85,B 0,C 180,E1 -3817.489,E2 -3817.489} C_VEL
LIN {X 0,Y 537.721,Z 255.887,A -85,B 0,C 180,E1 -3818.576,E2 -3818.576} C_VEL
LIN {X 0,Y 537.624,Z 261.516,A -85,B 0,C 180,E1 -3819.832,E2 -3819.832} C_VEL
LIN {X 0,Y 537.569,Z 264.966,A -85,B 0,C 180,E1 -3820.819,E2 -3820.819} C_VEL
LIN {X 0,Y 537.564,Z 267.635,A -85,B 0,C 180,E1 -3821.823,E2 -3821.823} C_VEL
LIN {X 0,Y 537.513,Z 269.718,A -85,B 0,C 180,E1 -3822.928,E2 -3822.928} C_VEL
LIN {X 0,Y 537.483,Z 270.915,A -85,B 0,C 180,E1 -3824.014,E2 -3824.014} C_VEL
LIN {X 0,Y 537.478,Z 271.301,A -85,B 0,C 180,E1 -3825.081,E2 -3825.081} C_VEL
LIN {X 0,Y 537.495,Z 270.875,A -85,B 0,C 180,E1 -3826.132,E2 -3826.132} C_VEL
LIN {X 0,Y 537.5,Z 269.707,A -85,B 0,C 180,E1 -3827.162,E2 -3827.162} C_VEL
LIN {X 0,Y 537.552,Z 266.624,A -85,B 0,C 180,E1 -3828.681,E2 -3828.681} C_VEL
LIN {X 0,Y 537.599,Z 263.409,A -85,B 0,C 180,E1 -3829.741,E2 -3829.741} C_VEL
LIN {X 0,Y 537.657,Z 259.232,A -85,B 0,C 180,E1 -3830.802,E2 -3830.802} C_VEL
LIN {X 0,Y 537.747,Z 253.951,A -85,B 0,C 180,E1 -3831.873,E2 -3831.873} C_VEL
LIN {X 0,Y 537.862,Z 246.684,A -85,B 0,C 180,E1 -3833.054,E2 -3833.054} C_VEL
LIN {X 0,Y 538.052,Z 238.844,A -85,B 0,C 180,E1 -3834.079,E2 -3834.079} C_VEL
LIN {X 0,Y 538.246,Z 229.771,A -85,B 0,C 180,E1 -3835.051,E2 -3835.051} C_VEL
LIN {X 0,Y 538.45,Z 219.311,A -85,B 0,C 180,E1 -3835.962,E2 -3835.962} C_VEL
LIN {X 0,Y 538.655,Z 207.505,A -85,B 0,C 180,E1 -3836.771,E2 -3836.771} C_VEL
LIN {X 0,Y 538.904,Z 195.687,A -85,B 0,C 180,E1 -3837.4,E2 -3837.4} C_VEL
LIN {X 0,Y 539.137,Z 183.106,A -85,B 0,C 180,E1 -3837.897,E2 -3837.897} C_VEL
LIN {X 0,Y 539.046,Z 176.635,A -85,B 0,C 180,E1 -3838.094,E2 -3838.094} C_VEL
LIN {X 0,Y 537.535,Z 168.627,A -85,B 0,C 180,E1 -3838.336,E2 -3838.336} C_VEL
LIN {X 0,Y 537.565,Z 165.326,A -85,B 0,C 180,E1 -3841.156,E2 -3841.156} C_VEL
LIN {X 0,Y 537.612,Z 162.487,A -85,B 0,C 180,E1 -3843.61,E2 -3843.61} C_VEL
LIN {X 0,Y 537.615,Z 159.451,A -85,B 0,C 180,E1 -3846.216,E2 -3846.216} C_VEL
LIN {X 0,Y 537.638,Z 156.785,A -85,B 0,C 180,E1 -3848.53,E2 -3848.53} C_VEL
LIN {X 0,Y 537.66,Z 154.003,A -85,B 0,C 180,E1 -3850.926,E2 -3850.926} C_VEL
LIN {X 0,Y 537.703,Z 151.292,A -85,B 0,C 180,E1 -3853.289,E2 -3853.289} C_VEL
LIN {X 0,Y 537.753,Z 148.564,A -85,B 0,C 180,E1 -3855.622,E2 -3855.622} C_VEL
LIN {X 0,Y 537.852,Z 145.492,A -85,B 0,C 180,E1 -3858.522,E2 -3858.522} C_VEL
LIN {X 0,Y 538.043,Z 145.465,A -85,B 0,C 180,E1 -3860.982,E2 -3860.982} C_VEL
LIN {X 0,Y 538.117,Z 145.459,A -85,B 0,C 180,E1 -3864.002,E2 -3864.002} C_VEL
LIN {X 0,Y 538.135,Z 145.453,A -85,B 0,C 180,E1 -3867.005,E2 -3867.005} C_VEL
LIN {X 0,Y 538.171,Z 145.452,A -85,B 0,C 180,E1 -3870,E2 -3870} C_VEL
LIN {X 0,Y 538.135,Z 145.452,A -85,B 0,C 180,E1 -3872.994,E2 -3872.994} C_VEL
LIN {X 0,Y 538.116,Z 145.459,A -85,B 0,C 180,E1 -3875.997,E2 -3875.997} C_VEL
LIN {X 0,Y 538.065,Z 145.461,A -85,B 0,C 180,E1 -3879.018,E2 -3879.018} C_VEL
LIN {X 0,Y 538.081,Z 145.463,A -85,B 0,C 180,E1 -3882.062,E2 -3882.062} C_VEL
LIN {X 0,Y 538.042,Z 145.465,A -85,B 0,C 180,E1 -3885.144,E2 -3885.144} C_VEL
LIN {X 0,Y 538.029,Z 145.467,A -85,B 0,C 180,E1 -3888.27,E2 -3888.27} C_VEL
LIN {X 0,Y 538.037,Z 145.468,A -85,B 0,C 180,E1 -3890.651,E2 -3890.651} C_VEL
LIN {X 0,Y 538.022,Z 145.469,A -85,B 0,C 180,E1 -3893.887,E2 -3893.887} C_VEL
LIN {X 0,Y 538.039,Z 145.467,A -85,B 0,C 180,E1 -3896.367,E2 -3896.367} C_VEL
LIN {X 0,Y 538.029,Z 145.469,A -85,B 0,C 180,E1 -3898.934,E2 -3898.934} C_VEL
LIN {X 0,Y 538.011,Z 145.469,A -85,B 0,C 180,E1 -3901.888,E2 -3901.888} C_VEL
LIN {X 0,Y 538.01,Z 145.469,A -85,B 0,C 180,E1 -3904.618,E2 -3904.618} C_VEL
LIN {X 0,Y 538.002,Z 145.472,A -85,B 0,C 180,E1 -3907.17,E2 -3907.17} C_VEL
LIN {X 0,Y 538.026,Z 145.469,A -85,B 0,C 180,E1 -3909.797,E2 -3909.797} C_VEL
LIN {X 0,Y 538.017,Z 145.468,A -85,B 0,C 180,E1 -3912.786,E2 -3912.786} C_VEL
LIN {X 0,Y 538.03,Z 145.467,A -85,B 0,C 180,E1 -3915.141,E2 -3915.141} C_VEL
LIN {X 0,Y 538.028,Z 145.469,A -85,B 0,C 180,E1 -3918.227,E2 -3918.227} C_VEL
LIN {X 0,Y 538.013,Z 145.469,A -85,B 0,C 180,E1 -3921.17,E2 -3921.17} C_VEL
LIN {X 0,Y 538.022,Z 145.468,A -85,B 0,C 180,E1 -3924.085,E2 -3924.085} C_VEL
LIN {X 0,Y 538.029,Z 145.47,A -85,B 0,C 180,E1 -3926.728,E2 -3926.728} C_VEL
LIN {X 0,Y 538.026,Z 145.466,A -85,B 0,C 180,E1 -3929.557,E2 -3929.557} C_VEL
LIN {X 0,Y 538.051,Z 145.467,A -85,B 0,C 180,E1 -3932.65,E2 -3932.65} C_VEL
LIN {X 0,Y 538.047,Z 145.466,A -85,B 0,C 180,E1 -3935.293,E2 -3935.293} C_VEL
LIN {X 0,Y 538.023,Z 145.469,A -85,B 0,C 180,E1 -3938.546,E2 -3938.546} C_VEL
LIN {X 0,Y 538.035,Z 145.468,A -85,B 0,C 180,E1 -3940.94,E2 -3940.94} C_VEL
LIN {X 0,Y 538.013,Z 145.469,A -85,B 0,C 180,E1 -3943.299,E2 -3943.299} C_VEL
LIN {X 0,Y 538.061,Z 145.462,A -85,B 0,C 180,E1 -3945.631,E2 -3945.631} C_VEL
LIN {X 0,Y 538.079,Z 145.461,A -85,B 0,C 180,E1 -3948.702,E2 -3948.702} C_VEL
LIN {X 0,Y 538.063,Z 145.463,A -85,B 0,C 180,E1 -3951.74,E2 -3951.74} C_VEL
LIN {X 0,Y 538.126,Z 145.455,A -85,B 0,C 180,E1 -3954.003,E2 -3954.003} C_VEL
LIN {X 0,Y 538.139,Z 145.455,A -85,B 0,C 180,E1 -3957.006,E2 -3957.006} C_VEL
LIN {X 0,Y 538.177,Z 145.449,A -85,B 0,C 180,E1 -3960,E2 -3960} C_VEL
LIN {X 0,Y 538.139,Z 145.455,A -85,B 0,C 180,E1 -3962.995,E2 -3962.995} C_VEL
LIN {X 0,Y 538.121,Z 145.456,A -85,B 0,C 180,E1 -3965.998,E2 -3965.998} C_VEL
LIN {X 0,Y 538.057,Z 145.465,A -85,B 0,C 180,E1 -3969.018,E2 -3969.018} C_VEL
LIN {X 0,Y 538.086,Z 145.46,A -85,B 0,C 180,E1 -3972.063,E2 -3972.063} C_VEL
LIN {X 0,Y 538.046,Z 145.467,A -85,B 0,C 180,E1 -3975.144,E2 -3975.144} C_VEL
LIN {X 0,Y 538.032,Z 145.467,A -85,B 0,C 180,E1 -3978.271,E2 -3978.271} C_VEL
LIN {X 0,Y 538.04,Z 145.465,A -85,B 0,C 180,E1 -3980.652,E2 -3980.652} C_VEL
LIN {X 0,Y 538.003,Z 145.47,A -85,B 0,C 180,E1 -3983.889,E2 -3983.889} C_VEL
LIN {X 0,Y 538.045,Z 145.464,A -85,B 0,C 180,E1 -3986.367,E2 -3986.367} C_VEL
LIN {X 0,Y 538.032,Z 145.466,A -85,B 0,C 180,E1 -3988.933,E2 -3988.933} C_VEL
LIN {X 0,Y 538.013,Z 145.471,A -85,B 0,C 180,E1 -3991.887,E2 -3991.887} C_VEL
LIN {X 0,Y 538.011,Z 145.47,A -85,B 0,C 180,E1 -3994.617,E2 -3994.617} C_VEL
LIN {X 0,Y 538.007,Z 145.47,A -85,B 0,C 180,E1 -3997.17,E2 -3997.17} C_VEL
LIN {X 0,Y 538.024,Z 145.467,A -85,B 0,C 180,E1 -3999.797,E2 -3999.797} C_VEL
LIN {X 0,Y 538.022,Z 145.469,A -85,B 0,C 180,E1 -4002.786,E2 -4002.786} C_VEL
LIN {X 0,Y 538.022,Z 145.466,A -85,B 0,C 180,E1 -4005.927,E2 -4005.927} C_VEL
LIN {X 0,Y 538.033,Z 145.465,A -85,B 0,C 180,E1 -4008.227,E2 -4008.227} C_VEL
LIN {X 0,Y 538.017,Z 145.471,A -85,B 0,C 180,E1 -4011.17,E2 -4011.17} C_VEL
LIN {X 0,Y 538.043,Z 145.566,A -85,B 0,C 180,E1 -4011.998,E2 -4011.998} C_VEL
LIN {X 0,Y 539.002,Z 151.266,A -85,B 0,C 180,E1 -4014.073,E2 -4014.073} C_VEL
LIN {X 0,Y 538.956,Z 158.524,A -85,B 0,C 180,E1 -4016.571,E2 -4016.571} C_VEL
LIN {X 0,Y 538.723,Z 167.141,A -85,B 0,C 180,E1 -4019.431,E2 -4019.431} C_VEL
LIN {X 0,Y 538.503,Z 176.863,A -85,B 0,C 180,E1 -4022.557,E2 -4022.557} C_VEL
LIN {X 0,Y 538.34,Z 185.634,A -85,B 0,C 180,E1 -4025.307,E2 -4025.307} C_VEL
LIN {X 0,Y 538.179,Z 194.408,A -85,B 0,C 180,E1 -4028,E2 -4028} C_VEL
LIN {X 0,Y 538.024,Z 202.844,A -85,B 0,C 180,E1 -4030.543,E2 -4030.543} C_VEL
LIN {X 0,Y 537.893,Z 212.112,A -85,B 0,C 180,E1 -4033.295,E2 -4033.295} C_VEL
LIN {X 0,Y 537.779,Z 221.379,A -85,B 0,C 180,E1 -4036.009,E2 -4036.009} C_VEL
LIN {X 0,Y 537.737,Z 223.53,A -85,B 0,C 180,E1 -4036.634,E2 -4036.634} C_VEL
LIN {X 0,Y 539.252,Z 234.356,A -85,B 0,C 180,E1 -4036.912,E2 -4036.912} C_VEL
LIN {X 0,Y 539.077,Z 246.477,A -85,B 0,C 180,E1 -4037.291,E2 -4037.291} C_VEL
LIN {X 0,Y 538.842,Z 257.489,A -85,B 0,C 180,E1 -4037.764,E2 -4037.764} C_VEL
LIN {X 0,Y 538.65,Z 268.431,A -85,B 0,C 180,E1 -4038.372,E2 -4038.372} C_VEL
LIN {X 0,Y 538.413,Z 279.927,A -85,B 0,C 180,E1 -4039.185,E2 -4039.185} C_VEL
LIN {X 0,Y 538.2,Z 289.602,A -85,B 0,C 180,E1 -4040.036,E2 -4040.036} C_VEL
LIN {X 0,Y 538.015,Z 298.414,A -85,B 0,C 180,E1 -4040.982,E2 -4040.982} C_VEL
LIN {X 0,Y 537.829,Z 307.002,A -85,B 0,C 180,E1 -4042.114,E2 -4042.114} C_VEL
LIN {X 0,Y 537.706,Z 313.868,A -85,B 0,C 180,E1 -4043.245,E2 -4043.245} C_VEL
LIN {X 0,Y 537.677,Z 319.366,A -85,B 0,C 180,E1 -4044.374,E2 -4044.374} C_VEL
LIN {X 0,Y 537.558,Z 323.678,A -85,B 0,C 180,E1 -4045.501,E2 -4045.501} C_VEL
LIN {X 0,Y 537.591,Z 325.958,A -85,B 0,C 180,E1 -4046.252,E2 -4046.252} C_VEL
LIN {X 0,Y 537.551,Z 327.808,A -85,B 0,C 180,E1 -4047.002,E2 -4047.002} C_VEL
LIN {X 0,Y 537.49,Z 329.198,A -85,B 0,C 180,E1 -4047.752,E2 -4047.752} C_VEL
LIN {X 0,Y 537.442,Z 330.785,A -85,B 0,C 180,E1 -4049.251,E2 -4049.251} C_VEL
LIN {X 0,Y 537.442,Z 331,A -85,B 0,C 180,E1 -4050,E2 -4050} C_VEL
LIN {X 0,Y 537.451,Z 330.186,A -85,B 0,C 180,E1 -4051.499,E2 -4051.499} C_VEL
LIN {X 0,Y 537.49,Z 329.199,A -85,B 0,C 180,E1 -4052.248,E2 -4052.248} C_VEL
LIN {X 0,Y 537.551,Z 327.81,A -85,B 0,C 180,E1 -4052.998,E2 -4052.998} C_VEL
LIN {X 0,Y 537.603,Z 324.895,A -85,B 0,C 180,E1 -4054.123,E2 -4054.123} C_VEL
LIN {X 0,Y 537.587,Z 320.948,A -85,B 0,C 180,E1 -4055.251,E2 -4055.251} C_VEL
LIN {X 0,Y 537.65,Z 316.099,A -85,B 0,C 180,E1 -4056.331,E2 -4056.331} C_VEL
LIN {X 0,Y 537.791,Z 309.468,A -85,B 0,C 180,E1 -4057.509,E2 -4057.509} C_VEL
LIN {X 0,Y 537.973,Z 301.477,A -85,B 0,C 180,E1 -4058.641,E2 -4058.641} C_VEL
LIN {X 0,Y 538.119,Z 293.334,A -85,B 0,C 180,E1 -4059.586,E2 -4059.586} C_VEL
LIN {X 0,Y 538.375,Z 283.399,A -85,B 0,C 180,E1 -4060.531,E2 -4060.531} C_VEL
LIN {X 0,Y 538.543,Z 273.584,A -85,B 0,C 180,E1 -4061.289,E2 -4061.289} C_VEL
LIN {X 0,Y 538.741,Z 262.592,A -85,B 0,C 180,E1 -4061.971,E2 -4061.971} C_VEL
LIN {X 0,Y 538.988,Z 250.106,A -85,B 0,C 180,E1 -4062.568,E2 -4062.568} C_VEL
LIN {X 0,Y 539.226,Z 237.083,A -85,B 0,C 180,E1 -4063.017,E2 -4063.017} C_VEL
LIN {X 0,Y 538.964,Z 230.928,A -85,B 0,C 180,E1 -4063.179,E2 -4063.179} C_VEL
LIN {X 0,Y 537.738,Z 223.53,A -85,B 0,C 180,E1 -4063.366,E2 -4063.366} C_VEL
LIN {X 0,Y 537.876,Z 213.435,A -85,B 0,C 180,E1 -4066.316,E2 -4066.316} C_VEL
LIN {X 0,Y 537.997,Z 204.167,A -85,B 0,C 180,E1 -4069.062,E2 -4069.062} C_VEL
LIN {X 0,Y 538.129,Z 196.224,A -85,B 0,C 180,E1 -4071.45,E2 -4071.45} C_VEL
LIN {X 0,Y 538.326,Z 186.958,A -85,B 0,C 180,E1 -4074.283,E2 -4074.283} C_VEL
LIN {X 0,Y 538.486,Z 177.689,A -85,B 0,C 180,E1 -4077.181,E2 -4077.181} C_VEL
LIN {X 0,Y 538.703,Z 168.443,A -85,B 0,C 180,E1 -4080.144,E2 -4080.144} C_VEL
LIN {X 0,Y 538.901,Z 159.056,A -85,B 0,C 180,E1 -4083.212,E2 -4083.212} C_VEL
LIN {X 0,Y 539.02,Z 152.307,A -85,B 0,C 180,E1 -4085.466,E2 -4085.466} C_VEL
LIN {X 0,Y 538.442,Z 147.57,A -85,B 0,C 180,E1 -4087.231,E2 -4087.231} C_VEL
LIN {X 0,Y 538.018,Z 145.471,A -85,B 0,C 180,E1 -4088.133,E2 -4088.133} C_VEL
LIN {X 0,Y 538.053,Z 145.466,A -85,B 0,C 180,E1 -4090.776,E2 -4090.776} C_VEL
LIN {X 0,Y 538.035,Z 145.468,A -85,B 0,C 180,E1 -4094.075,E2 -4094.075} C_VEL
LIN {X 0,Y 538.03,Z 145.469,A -85,B 0,C 180,E1 -4097.012,E2 -4097.012} C_VEL
LIN {X 0,Y 538.056,Z 145.468,A -85,B 0,C 180,E1 -4099.252,E2 -4099.252} C_VEL
LIN {X 0,Y 537.997,Z 145.474,A -85,B 0,C 180,E1 -4102.122,E2 -4102.122} C_VEL
LIN {X 0,Y 538.005,Z 145.471,A -85,B 0,C 180,E1 -4104.916,E2 -4104.916} C_VEL
LIN {X 0,Y 538.032,Z 145.468,A -85,B 0,C 180,E1 -4107.618,E2 -4107.618} C_VEL
LIN {X 0,Y 538.023,Z 145.47,A -85,B 0,C 180,E1 -4110.239,E2 -4110.239} C_VEL
LIN {X 0,Y 538.068,Z 145.462,A -85,B 0,C 180,E1 -4112.796,E2 -4112.796} C_VEL
LIN {X 0,Y 538.053,Z 145.466,A -85,B 0,C 180,E1 -4115.292,E2 -4115.292} C_VEL
LIN {X 0,Y 538.027,Z 145.47,A -85,B 0,C 180,E1 -4118.546,E2 -4118.546} C_VEL
LIN {X 0,Y 538.038,Z 145.467,A -85,B 0,C 180,E1 -4120.94,E2 -4120.94} C_VEL
LIN {X 0,Y 538.017,Z 145.47,A -85,B 0,C 180,E1 -4123.298,E2 -4123.298} C_VEL
LIN {X 0,Y 538.069,Z 145.464,A -85,B 0,C 180,E1 -4125.63,E2 -4125.63} C_VEL
LIN {X 0,Y 538.083,Z 145.462,A -85,B 0,C 180,E1 -4128.701,E2 -4128.701} C_VEL
LIN {X 0,Y 538.091,Z 145.461,A -85,B 0,C 180,E1 -4131.739,E2 -4131.739} C_VEL
LIN {X 0,Y 538.166,Z 145.452,A -85,B 0,C 180,E1 -4134.755,E2 -4134.755} C_VEL
LIN {X 0,Y 538.173,Z 145.451,A -85,B 0,C 180,E1 -4137.754,E2 -4137.754} C_VEL
LIN {X 0,Y 538.188,Z 145.449,A -85,B 0,C 180,E1 -4140.748,E2 -4140.748} C_VEL
LIN {X 0,Y 538.141,Z 145.454,A -85,B 0,C 180,E1 -4142.994,E2 -4142.994} C_VEL
LIN {X 0,Y 538.126,Z 145.457,A -85,B 0,C 180,E1 -4145.997,E2 -4145.997} C_VEL
LIN {X 0,Y 538.083,Z 145.462,A -85,B 0,C 180,E1 -4148.26,E2 -4148.26} C_VEL
LIN {X 0,Y 537.92,Z 145.485,A -85,B 0,C 180,E1 -4150.539,E2 -4150.539} C_VEL
LIN {X 0,Y 537.854,Z 145.891,A -85,B 0,C 180,E1 -4151.475,E2 -4151.475} C_VEL
LIN {X 0,Y 537.824,Z 149.674,A -85,B 0,C 180,E1 -4154.761,E2 -4154.761} C_VEL
LIN {X 0,Y 537.758,Z 152.786,A -85,B 0,C 180,E1 -4157.493,E2 -4157.493} C_VEL
LIN {X 0,Y 537.668,Z 156.289,A -85,B 0,C 180,E1 -4160.666,E2 -4160.666} C_VEL
LIN {X 0,Y 537.621,Z 159.854,A -85,B 0,C 180,E1 -4163.784,E2 -4163.784} C_VEL
LIN {X 0,Y 537.636,Z 162.77,A -85,B 0,C 180,E1 -4166.388,E2 -4166.388} C_VEL
LIN {X 0,Y 537.594,Z 165.623,A -85,B 0,C 180,E1 -4168.927,E2 -4168.927} C_VEL
LIN {X 0,Y 537.574,Z 168.856,A -85,B 0,C 180,E1 -4171.767,E2 -4171.767} C_VEL
LIN {X 0,Y 539.214,Z 178.488,A -85,B 0,C 180,E1 -4172.047,E2 -4172.047} C_VEL
LIN {X 0,Y 539.006,Z 190.983,A -85,B 0,C 180,E1 -4172.482,E2 -4172.482} C_VEL
LIN {X 0,Y 538.786,Z 203.97,A -85,B 0,C 180,E1 -4173.108,E2 -4173.108} C_VEL
LIN {X 0,Y 538.539,Z 215.343,A -85,B 0,C 180,E1 -4173.828,E2 -4173.828} C_VEL
LIN {X 0,Y 538.422,Z 223.494,A -85,B 0,C 180,E1 -4174.463,E2 -4174.463} C_VEL
LIN {X 0,Y 537.66,Z 228.095,A -85,B 0,C 180,E1 -4174.85,E2 -4174.85} C_VEL
LIN {X 0,Y 534.663,Z 235.298,A -85,B 0,C 180,E1 -4175.506,E2 -4175.506} C_VEL
LIN {X 0,Y 531.65,Z 241.939,A -85,B 0,C 180,E1 -4176.228,E2 -4176.228} C_VEL
LIN {X 0,Y 530.87,Z 245.658,A -85,B 0,C 180,E1 -4176.716,E2 -4176.716} C_VEL
LIN {X 0,Y 530.764,Z 252.367,A -85,B 0,C 180,E1 -4177.763,E2 -4177.763} C_VEL
LIN {X 0,Y 530.62,Z 258.811,A -85,B 0,C 180,E1 -4179.014,E2 -4179.014} C_VEL
LIN {X 0,Y 530.535,Z 263.224,A -85,B 0,C 180,E1 -4180.108,E2 -4180.108} C_VEL
LIN {X 0,Y 530.495,Z 267.38,A -85,B 0,C 180,E1 -4181.483,E2 -4181.483} C_VEL
LIN {X 0,Y 530.429,Z 269.544,A -85,B 0,C 180,E1 -4182.51,E2 -4182.51} C_VEL
LIN {X 0,Y 530.404,Z 270.958,A -85,B 0,C 180,E1 -4183.551,E2 -4183.551} C_VEL
LIN {X 0,Y 530.404,Z 271.65,A -85,B 0,C 180,E1 -4184.608,E2 -4184.608} C_VEL
LIN {X 0,Y 530.405,Z 271.59,A -85,B 0,C 180,E1 -4185.685,E2 -4185.685} C_VEL
LIN {X 0,Y 530.409,Z 270.689,A -85,B 0,C 180,E1 -4186.782,E2 -4186.782} C_VEL
LIN {X 0,Y 530.451,Z 268.92,A -85,B 0,C 180,E1 -4187.897,E2 -4187.897} C_VEL
LIN {X 0,Y 530.498,Z 266.194,A -85,B 0,C 180,E1 -4189.036,E2 -4189.036} C_VEL
LIN {X 0,Y 530.578,Z 262.383,A -85,B 0,C 180,E1 -4190.197,E2 -4190.197} C_VEL
LIN {X 0,Y 530.672,Z 256.736,A -85,B 0,C 180,E1 -4191.505,E2 -4191.505} C_VEL
LIN {X 0,Y 530.798,Z 249.324,A -85,B 0,C 180,E1 -4192.816,E2 -4192.816} C_VEL
LIN {X 0,Y 530.988,Z 241.032,A -85,B 0,C 180,E1 -4193.98,E2 -4193.98} C_VEL
LIN {X 0,Y 531.23,Z 232.197,A -85,B 0,C 180,E1 -4194.98,E2 -4194.98} C_VEL
LIN {X 0,Y 531.455,Z 221.957,A -85,B 0,C 180,E1 -4195.918,E2 -4195.918} C_VEL
LIN {X 0,Y 531.692,Z 210.919,A -85,B 0,C 180,E1 -4196.732,E2 -4196.732} C_VEL
LIN {X 0,Y 531.886,Z 200.559,A -85,B 0,C 180,E1 -4197.34,E2 -4197.34} C_VEL
LIN {X 0,Y 532.202,Z 187.98,A -85,B 0,C 180,E1 -4197.9,E2 -4197.9} C_VEL
LIN {X 0,Y 532.139,Z 177.549,A -85,B 0,C 180,E1 -4198.249,E2 -4198.249} C_VEL
LIN {X 0,Y 530.44,Z 169.038,A -85,B 0,C 180,E1 -4198.512,E2 -4198.512} C_VEL
LIN {X 0,Y 530.484,Z 165.529,A -85,B 0,C 180,E1 -4201.514,E2 -4201.514} C_VEL
LIN {X 0,Y 530.555,Z 162.32,A -85,B 0,C 180,E1 -4204.257,E2 -4204.257} C_VEL
LIN {X 0,Y 530.541,Z 159.638,A -85,B 0,C 180,E1 -4206.584,E2 -4206.584} C_VEL
LIN {X 0,Y 530.558,Z 156.799,A -85,B 0,C 180,E1 -4209.044,E2 -4209.044} C_VEL
LIN {X 0,Y 530.569,Z 154.027,A -85,B 0,C 180,E1 -4211.463,E2 -4211.463} C_VEL
LIN {X 0,Y 530.633,Z 151.252,A -85,B 0,C 180,E1 -4213.851,E2 -4213.851} C_VEL
LIN {X 0,Y 530.661,Z 148.573,A -85,B 0,C 180,E1 -4216.208,E2 -4216.208} C_VEL
LIN {X 0,Y 530.706,Z 146.791,A -85,B 0,C 180,E1 -4217.767,E2 -4217.767} C_VEL
LIN {X 0,Y 530.818,Z 146.368,A -85,B 0,C 180,E1 -4218.545,E2 -4218.545} C_VEL
LIN {X 0,Y 531.046,Z 146.339,A -85,B 0,C 180,E1 -4221.629,E2 -4221.629} C_VEL
LIN {X 0,Y 531.118,Z 146.328,A -85,B 0,C 180,E1 -4224.685,E2 -4224.685} C_VEL
LIN {X 0,Y 531.14,Z 146.327,A -85,B 0,C 180,E1 -4227.725,E2 -4227.725} C_VEL
LIN {X 0,Y 531.149,Z 146.324,A -85,B 0,C 180,E1 -4230.758,E2 -4230.758} C_VEL
LIN {X 0,Y 531.102,Z 146.328,A -85,B 0,C 180,E1 -4233.034,E2 -4233.034} C_VEL
LIN {X 0,Y 531.071,Z 146.336,A -85,B 0,C 180,E1 -4236.077,E2 -4236.077} C_VEL
LIN {X 0,Y 531.052,Z 146.338,A -85,B 0,C 180,E1 -4238.37,E2 -4238.37} C_VEL
LIN {X 0,Y 531.049,Z 146.337,A -85,B 0,C 180,E1 -4241.672,E2 -4241.672} C_VEL
LIN {X 0,Y 531.028,Z 146.339,A -85,B 0,C 180,E1 -4244.956,E2 -4244.956} C_VEL
LIN {X 0,Y 531.014,Z 146.342,A -85,B 0,C 180,E1 -4247.722,E2 -4247.722} C_VEL
LIN {X 0,Y 530.997,Z 146.343,A -85,B 0,C 180,E1 -4250.938,E2 -4250.938} C_VEL
LIN {X 0,Y 530.977,Z 146.346,A -85,B 0,C 180,E1 -4254.225,E2 -4254.225} C_VEL
LIN {X 0,Y 531.001,Z 146.344,A -85,B 0,C 180,E1 -4256.744,E2 -4256.744} C_VEL
LIN {X 0,Y 530.98,Z 146.346,A -85,B 0,C 180,E1 -4259.323,E2 -4259.323} C_VEL
LIN {X 0,Y 530.967,Z 146.346,A -85,B 0,C 180,E1 -4262.101,E2 -4262.101} C_VEL
LIN {X 0,Y 530.968,Z 146.348,A -85,B 0,C 180,E1 -4264.851,E2 -4264.851} C_VEL
LIN {X 0,Y 530.963,Z 146.349,A -85,B 0,C 180,E1 -4267.508,E2 -4267.508} C_VEL
LIN {X 0,Y 530.982,Z 146.344,A -85,B 0,C 180,E1 -4270.433,E2 -4270.433} C_VEL
LIN {X 0,Y 530.963,Z 146.349,A -85,B 0,C 180,E1 -4273.495,E2 -4273.495} C_VEL
LIN {X 0,Y 530.963,Z 146.347,A -85,B 0,C 180,E1 -4276.506,E2 -4276.506} C_VEL
LIN {X 0,Y 530.979,Z 146.346,A -85,B 0,C 180,E1 -4279.567,E2 -4279.567} C_VEL
LIN {X 0,Y 530.967,Z 146.347,A -85,B 0,C 180,E1 -4282.577,E2 -4282.577} C_VEL
LIN {X 0,Y 530.993,Z 146.345,A -85,B 0,C 180,E1 -4285.311,E2 -4285.311} C_VEL
LIN {X 0,Y 530.966,Z 146.349,A -85,B 0,C 180,E1 -4288.032,E2 -4288.032} C_VEL
LIN {X 0,Y 530.988,Z 146.344,A -85,B 0,C 180,E1 -4290.875,E2 -4290.875} C_VEL
LIN {X 0,Y 531.001,Z 146.342,A -85,B 0,C 180,E1 -4293.257,E2 -4293.257} C_VEL
LIN {X 0,Y 530.984,Z 146.344,A -85,B 0,C 180,E1 -4295.961,E2 -4295.961} C_VEL
LIN {X 0,Y 531,Z 146.342,A -85,B 0,C 180,E1 -4299.063,E2 -4299.063} C_VEL
LIN {X 0,Y 530.986,Z 146.345,A -85,B 0,C 180,E1 -4301.479,E2 -4301.479} C_VEL
LIN {X 0,Y 530.995,Z 146.345,A -85,B 0,C 180,E1 -4304.651,E2 -4304.651} C_VEL
LIN {X 0,Y 531.041,Z 146.337,A -85,B 0,C 180,E1 -4307.776,E2 -4307.776} C_VEL
LIN {X 0,Y 531.026,Z 146.341,A -85,B 0,C 180,E1 -4310.862,E2 -4310.862} C_VEL
LIN {X 0,Y 531.086,Z 146.332,A -85,B 0,C 180,E1 -4313.923,E2 -4313.923} C_VEL
LIN {X 0,Y 531.106,Z 146.331,A -85,B 0,C 180,E1 -4316.966,E2 -4316.966} C_VEL
LIN {X 0,Y 531.147,Z 146.324,A -85,B 0,C 180,E1 -4320,E2 -4320} C_VEL
LIN {X 0,Y 531.106,Z 146.331,A -85,B 0,C 180,E1 -4323.035,E2 -4323.035} C_VEL
LIN {X 0,Y 531.075,Z 146.333,A -85,B 0,C 180,E1 -4326.078,E2 -4326.078} C_VEL
LIN {X 0,Y 531.019,Z 146.342,A -85,B 0,C 180,E1 -4329.139,E2 -4329.139} C_VEL
LIN {X 0,Y 531.043,Z 146.338,A -85,B 0,C 180,E1 -4332.225,E2 -4332.225} C_VEL
LIN {X 0,Y 530.996,Z 146.344,A -85,B 0,C 180,E1 -4335.35,E2 -4335.35} C_VEL
LIN {X 0,Y 530.99,Z 146.345,A -85,B 0,C 180,E1 -4338.522,E2 -4338.522} C_VEL
LIN {X 0,Y 531.001,Z 146.343,A -85,B 0,C 180,E1 -4340.938,E2 -4340.938} C_VEL
LIN {X 0,Y 530.973,Z 146.346,A -85,B 0,C 180,E1 -4344.225,E2 -4344.225} C_VEL
LIN {X 0,Y 531.005,Z 146.341,A -85,B 0,C 180,E1 -4346.744,E2 -4346.744} C_VEL
LIN {X 0,Y 530.983,Z 146.346,A -85,B 0,C 180,E1 -4349.323,E2 -4349.323} C_VEL
LIN {X 0,Y 530.967,Z 146.347,A -85,B 0,C 180,E1 -4352.1,E2 -4352.1} C_VEL
LIN {X 0,Y 530.97,Z 146.346,A -85,B 0,C 180,E1 -4354.851,E2 -4354.851} C_VEL
LIN {X 0,Y 530.968,Z 146.347,A -85,B 0,C 180,E1 -4357.508,E2 -4357.508} C_VEL
LIN {X 0,Y 530.983,Z 146.347,A -85,B 0,C 180,E1 -4360.433,E2 -4360.433} C_VEL
LIN {X 0,Y 530.963,Z 146.345,A -85,B 0,C 180,E1 -4363.281,E2 -4363.281} C_VEL
LIN {X 0,Y 530.984,Z 146.342,A -85,B 0,C 180,E1 -4365.622,E2 -4365.622} C_VEL
LIN {X 0,Y 530.996,Z 146.343,A -85,B 0,C 180,E1 -4368.565,E2 -4368.565} C_VEL
LIN {X 0,Y 530.999,Z 146.407,A -85,B 0,C 180,E1 -4371.714,E2 -4371.714} C_VEL
LIN {X 0,Y 532.054,Z 152.776,A -85,B 0,C 180,E1 -4374.09,E2 -4374.09} C_VEL
LIN {X 0,Y 532.013,Z 159.28,A -85,B 0,C 180,E1 -4376.33,E2 -4376.33} C_VEL
LIN {X 0,Y 531.772,Z 167.818,A -85,B 0,C 180,E1 -4379.211,E2 -4379.211} C_VEL
LIN {X 0,Y 531.526,Z 177.69,A -85,B 0,C 180,E1 -4382.433,E2 -4382.433} C_VEL
LIN {X 0,Y 531.327,Z 186.958,A -85,B 0,C 180,E1 -4385.376,E2 -4385.376} C_VEL
LIN {X 0,Y 531.118,Z 196.225,A -85,B 0,C 180,E1 -4388.253,E2 -4388.253} C_VEL
LIN {X 0,Y 530.959,Z 205.492,A -85,B 0,C 180,E1 -4391.077,E2 -4391.077} C_VEL
LIN {X 0,Y 530.814,Z 214.76,A -85,B 0,C 180,E1 -4393.857,E2 -4393.857} C_VEL
LIN {X 0,Y 530.696,Z 223.53,A -85,B 0,C 180,E1 -4396.454,E2 -4396.454} C_VEL
LIN {X 0,Y 532.35,Z 234.356,A -85,B 0,C 180,E1 -4396.739,E2 -4396.739} C_VEL
LIN {X 0,Y 532.142,Z 246.477,A -85,B 0,C 180,E1 -4397.123,E2 -4397.123} C_VEL
LIN {X 0,Y 531.902,Z 257.49,A -85,B 0,C 180,E1 -4397.602,E2 -4397.602} C_VEL
LIN {X 0,Y 531.688,Z 269.006,A -85,B 0,C 180,E1 -4398.253,E2 -4398.253} C_VEL
LIN {X 0,Y 531.43,Z 279.926,A -85,B 0,C 180,E1 -4399.041,E2 -4399.041} C_VEL
LIN {X 0,Y 531.192,Z 289.602,A -85,B 0,C 180,E1 -4399.904,E2 -4399.904} C_VEL
LIN {X 0,Y 530.969,Z 298.414,A -85,B 0,C 180,E1 -4400.861,E2 -4400.861} C_VEL
LIN {X 0,Y 530.78,Z 307.002,A -85,B 0,C 180,E1 -4402.008,E2 -4402.008} C_VEL
LIN {X 0,Y 530.637,Z 313.869,A -85,B 0,C 180,E1 -4403.154,E2 -4403.154} C_VEL
LIN {X 0,Y 530.611,Z 319.366,A -85,B 0,C 180,E1 -4404.299,E2 -4404.299} C_VEL
LIN {X 0,Y 530.457,Z 323.678,A -85,B 0,C 180,E1 -4405.441,E2 -4405.441} C_VEL
LIN {X 0,Y 530.516,Z 325.958,A -85,B 0,C 180,E1 -4406.202,E2 -4406.202} C_VEL
LIN {X 0,Y 530.457,Z 327.808,A -85,B 0,C 180,E1 -4406.962,E2 -4406.962} C_VEL
LIN {X 0,Y 530.411,Z 329.198,A -85,B 0,C 180,E1 -4407.722,E2 -4407.722} C_VEL
LIN {X 0,Y 530.344,Z 330.785,A -85,B 0,C 180,E1 -4409.241,E2 -4409.241} C_VEL
LIN {X 0,Y 530.342,Z 331,A -85,B 0,C 180,E1 -4410,E2 -4410} C_VEL
LIN {X 0,Y 530.361,Z 330.186,A -85,B 0,C 180,E1 -4411.519,E2 -4411.519} C_VEL
LIN {X 0,Y 530.412,Z 329.199,A -85,B 0,C 180,E1 -4412.278,E2 -4412.278} C_VEL
LIN {X 0,Y 530.457,Z 327.81,A -85,B 0,C 180,E1 -4413.038,E2 -4413.038} C_VEL
LIN {X 0,Y 530.523,Z 324.895,A -85,B 0,C 180,E1 -4414.178,E2 -4414.178} C_VEL
LIN {X 0,Y 530.525,Z 320.948,A -85,B 0,C 180,E1 -4415.321,E2 -4415.321} C_VEL
LIN {X 0,Y 530.599,Z 315.267,A -85,B 0,C 180,E1 -4416.581,E2 -4416.581} C_VEL
LIN {X 0,Y 530.759,Z 308.236,A -85,B 0,C 180,E1 -4417.801,E2 -4417.801} C_VEL
LIN {X 0,Y 530.931,Z 299.989,A -85,B 0,C 180,E1 -4418.948,E2 -4418.948} C_VEL
LIN {X 0,Y 531.113,Z 291.537,A -85,B 0,C 180,E1 -4419.906,E2 -4419.906} C_VEL
LIN {X 0,Y 531.398,Z 281.096,A -85,B 0,C 180,E1 -4420.863,E2 -4420.863} C_VEL
LIN {X 0,Y 531.642,Z 269.312,A -85,B 0,C 180,E1 -4421.728,E2 -4421.728} C_VEL
LIN {X 0,Y 531.905,Z 257.483,A -85,B 0,C 180,E1 -4422.399,E2 -4422.399} C_VEL
LIN {X 0,Y 532.151,Z 245.165,A -85,B 0,C 180,E1 -4422.926,E2 -4422.926} C_VEL
LIN {X 0,Y 532.218,Z 232.969,A -85,B 0,C 180,E1 -4423.301,E2 -4423.301} C_VEL
LIN {X 0,Y 530.696,Z 223.53,A -85,B 0,C 180,E1 -4423.547,E2 -4423.547} C_VEL
LIN {X 0,Y 530.815,Z 214.759,A -85,B 0,C 180,E1 -4426.143,E2 -4426.143} C_VEL
LIN {X 0,Y 530.96,Z 205.491,A -85,B 0,C 180,E1 -4428.923,E2 -4428.923} C_VEL
LIN {X 0,Y 531.119,Z 196.224,A -85,B 0,C 180,E1 -4431.747,E2 -4431.747} C_VEL
LIN {X 0,Y 531.327,Z 186.957,A -85,B 0,C 180,E1 -4434.624,E2 -4434.624} C_VEL
LIN {X 0,Y 531.522,Z 177.474,A -85,B 0,C 180,E1 -4437.637,E2 -4437.637} C_VEL
LIN {X 0,Y 531.756,Z 167.789,A -85,B 0,C 180,E1 -4440.786,E2 -4440.786} C_VEL
LIN {X 0,Y 531.983,Z 158.966,A -85,B 0,C 180,E1 -4443.701,E2 -4443.701} C_VEL
LIN {X 0,Y 532.078,Z 153.565,A -85,B 0,C 180,E1 -4445.534,E2 -4445.534} C_VEL
LIN {X 0,Y 531.404,Z 148.48,A -85,B 0,C 180,E1 -4447.484,E2 -4447.484} C_VEL
LIN {X 0,Y 530.985,Z 146.347,A -85,B 0,C 180,E1 -4448.347,E2 -4448.347} C_VEL
LIN {X 0,Y 531.001,Z 146.345,A -85,B 0,C 180,E1 -4451.435,E2 -4451.435} C_VEL
LIN {X 0,Y 530.993,Z 146.345,A -85,B 0,C 180,E1 -4454.547,E2 -4454.547} C_VEL
LIN {X 0,Y 530.988,Z 146.346,A -85,B 0,C 180,E1 -4457.834,E2 -4457.834} C_VEL
LIN {X 0,Y 530.993,Z 146.346,A -85,B 0,C 180,E1 -4460.557,E2 -4460.557} C_VEL
LIN {X 0,Y 530.96,Z 146.35,A -85,B 0,C 180,E1 -4463.441,E2 -4463.441} C_VEL
LIN {X 0,Y 531.004,Z 146.344,A -85,B 0,C 180,E1 -4466.494,E2 -4466.494} C_VEL
LIN {X 0,Y 530.979,Z 146.347,A -85,B 0,C 180,E1 -4469.355,E2 -4469.355} C_VEL
LIN {X 0,Y 531.02,Z 146.342,A -85,B 0,C 180,E1 -4472.467,E2 -4472.467} C_VEL
LIN {X 0,Y 531.01,Z 146.342,A -85,B 0,C 180,E1 -4474.942,E2 -4474.942} C_VEL
LIN {X 0,Y 530.976,Z 146.347,A -85,B 0,C 180,E1 -4478.247,E2 -4478.247} C_VEL
LIN {X 0,Y 530.997,Z 146.345,A -85,B 0,C 180,E1 -4480.677,E2 -4480.677} C_VEL
LIN {X 0,Y 530.975,Z 146.346,A -85,B 0,C 180,E1 -4483.07,E2 -4483.07} C_VEL
LIN {X 0,Y 531.025,Z 146.342,A -85,B 0,C 180,E1 -4485.436,E2 -4485.436} C_VEL
LIN {X 0,Y 531.042,Z 146.34,A -85,B 0,C 180,E1 -4488.549,E2 -4488.549} C_VEL
LIN {X 0,Y 531.06,Z 146.338,A -85,B 0,C 180,E1 -4491.629,E2 -4491.629} C_VEL
LIN {X 0,Y 531.125,Z 146.329,A -85,B 0,C 180,E1 -4494.685,E2 -4494.685} C_VEL
LIN {X 0,Y 531.145,Z 146.327,A -85,B 0,C 180,E1 -4497.725,E2 -4497.725} C_VEL
LIN {X 0,Y 531.158,Z 146.325,A -85,B 0,C 180,E1 -4500.758,E2 -4500.758} C_VEL
LIN {X 0,Y 531.108,Z 146.33,A -85,B 0,C 180,E1 -4503.034,E2 -4503.034} C_VEL
LIN {X 0,Y 531.086,Z 146.334,A -85,B 0,C 180,E1 -4506.077,E2 -4506.077} C_VEL
LIN {X 0,Y 531.051,Z 146.338,A -85,B 0,C 180,E1 -4508.37,E2 -4508.37} C_VEL
LIN {X 0,Y 530.857,Z 146.365,A -85,B 0,C 180,E1 -4510.681,E2 -4510.681} C_VEL
LIN {X 0,Y 530.808,Z 146.731,A -85,B 0,C 180,E1 -4511.542,E2 -4511.542} C_VEL
LIN {X 0,Y 530.764,Z 150.496,A -85,B 0,C 180,E1 -4514.846,E2 -4514.846} C_VEL
LIN {X 0,Y 530.69,Z 153.763,A -85,B 0,C 180,E1 -4517.733,E2 -4517.733} C_VEL
LIN {X 0,Y 530.615,Z 157.366,A -85,B 0,C 180,E1 -4520.953,E2 -4520.953} C_VEL
LIN {X 0,Y 530.552,Z 160.666,A -85,B 0,C 180,E1 -4523.933,E2 -4523.933} C_VEL
LIN {X 0,Y 530.561,Z 163.872,A -85,B 0,C 180,E1 -4526.767,E2 -4526.767} C_VEL
LIN {X 0,Y 530.513,Z 166.788,A -85,B 0,C 180,E1 -4529.351,E2 -4529.351} C_VEL
LIN {X 0,Y 530.509,Z 169.324,A -85,B 0,C 180,E1 -4531.58,E2 -4531.58} C_VEL
LIN {X 0,Y 532.31,Z 179.336,A -85,B 0,C 180,E1 -4531.891,E2 -4531.891} C_VEL
LIN {X 0,Y 532.1,Z 191.979,A -85,B 0,C 180,E1 -4532.343,E2 -4532.343} C_VEL
LIN {X 0,Y 531.876,Z 203.711,A -85,B 0,C 180,E1 -4532.916,E2 -4532.916} C_VEL
LIN {X 0,Y 531.596,Z 214.669,A -85,B 0,C 180,E1 -4533.602,E2 -4533.602} C_VEL
LIN {X 0,Y 531.425,Z 225.092,A -85,B 0,C 180,E1 -4534.427,E2 -4534.427} C_VEL
LIN {X 0,Y 531.183,Z 235.112,A -85,B 0,C 180,E1 -4535.409,E2 -4535.409} C_VEL
LIN {X 0,Y 530.955,Z 242.787,A -85,B 0,C 180,E1 -4536.326,E2 -4536.326} C_VEL
LIN {X 0,Y 530.87,Z 245.658,A -85,B 0,C 180,E1 -4536.716,E2 -4536.716} C_VEL
LIN {X 0,Y 530.1,Z 249.211,A -85,B 0,C 180,E1 -4537.225,E2 -4537.225} C_VEL
LIN {X 0,Y 527.126,Z 254.595,A -85,B 0,C 180,E1 -4538.072,E2 -4538.072} C_VEL
LIN {X 0,Y 524.204,Z 259.328,A -85,B 0,C 180,E1 -4538.967,E2 -4538.967} C_VEL
LIN {X 0,Y 523.519,Z 261.817,A -85,B 0,C 180,E1 -4539.545,E2 -4539.545} C_VEL
LIN {X 0,Y 523.441,Z 265.593,A -85,B 0,C 180,E1 -4540.631,E2 -4540.631} C_VEL
LIN {X 0,Y 523.395,Z 268.374,A -85,B 0,C 180,E1 -4541.679,E2 -4541.679} C_VEL
LIN {X 0,Y 523.349,Z 271.075,A -85,B 0,C 180,E1 -4543.225,E2 -4543.225} C_VEL
LIN {X 0,Y 523.317,Z 272.085,A -85,B 0,C 180,E1 -4544.62,E2 -4544.62} C_VEL
LIN {X 0,Y 523.318,Z 272.012,A -85,B 0,C 180,E1 -4545.705,E2 -4545.705} C_VEL
LIN {X 0,Y 523.324,Z 271.149,A -85,B 0,C 180,E1 -4546.771,E2 -4546.771} C_VEL
LIN {X 0,Y 523.368,Z 269.551,A -85,B 0,C 180,E1 -4547.823,E2 -4547.823} C_VEL
LIN {X 0,Y 523.415,Z 267.245,A -85,B 0,C 180,E1 -4548.857,E2 -4548.857} C_VEL
LIN {X 0,Y 523.466,Z 264.02,A -85,B 0,C 180,E1 -4549.931,E2 -4549.931} C_VEL
LIN {X 0,Y 523.556,Z 259.293,A -85,B 0,C 180,E1 -4551.129,E2 -4551.129} C_VEL
LIN {X 0,Y 523.667,Z 253.094,A -85,B 0,C 180,E1 -4552.356,E2 -4552.356} C_VEL
LIN {X 0,Y 523.893,Z 245.166,A -85,B 0,C 180,E1 -4553.599,E2 -4553.599} C_VEL
LIN {X 0,Y 524.153,Z 236.626,A -85,B 0,C 180,E1 -4554.673,E2 -4554.673} C_VEL
LIN {X 0,Y 524.359,Z 227.324,A -85,B 0,C 180,E1 -4555.625,E2 -4555.625} C_VEL
LIN {X 0,Y 524.58,Z 216.761,A -85,B 0,C 180,E1 -4556.503,E2 -4556.503} C_VEL
LIN {X 0,Y 524.853,Z 205.549,A -85,B 0,C 180,E1 -4557.246,E2 -4557.246} C_VEL
LIN {X 0,Y 525.159,Z 193.404,A -85,B 0,C 180,E1 -4557.862,E2 -4557.862} C_VEL
LIN {X 0,Y 525.389,Z 180.055,A -85,B 0,C 180,E1 -4558.357,E2 -4558.357} C_VEL
LIN {X 0,Y 523.703,Z 171.072,A -85,B 0,C 180,E1 -4558.636,E2 -4558.636} C_VEL
LIN {X 0,Y 523.395,Z 169.409,A -85,B 0,C 180,E1 -4558.699,E2 -4558.699} C_VEL
LIN {X 0,Y 523.41,Z 166.615,A -85,B 0,C 180,E1 -4561.093,E2 -4561.093} C_VEL
LIN {X 0,Y 523.506,Z 163.127,A -85,B 0,C 180,E1 -4564.087,E2 -4564.087} C_VEL
LIN {X 0,Y 523.455,Z 159.669,A -85,B 0,C 180,E1 -4567.085,E2 -4567.085} C_VEL
LIN {X 0,Y 523.51,Z 156.34,A -85,B 0,C 180,E1 -4570.006,E2 -4570.006} C_VEL
LIN {X 0,Y 523.59,Z 153.097,A -85,B 0,C 180,E1 -4572.824,E2 -4572.824} C_VEL
LIN {X 0,Y 523.65,Z 150.352,A -85,B 0,C 180,E1 -4575.226,E2 -4575.226} C_VEL
LIN {X 0,Y 523.646,Z 147.672,A -85,B 0,C 180,E1 -4577.6,E2 -4577.6} C_VEL
LIN {X 0,Y 523.758,Z 147.247,A -85,B 0,C 180,E1 -4578.388,E2 -4578.388} C_VEL
LIN {X 0,Y 523.992,Z 147.217,A -85,B 0,C 180,E1 -4581.516,E2 -4581.516} C_VEL
LIN {X 0,Y 524.079,Z 147.205,A -85,B 0,C 180,E1 -4584.613,E2 -4584.613} C_VEL
LIN {X 0,Y 524.111,Z 147.203,A -85,B 0,C 180,E1 -4587.694,E2 -4587.694} C_VEL
LIN {X 0,Y 524.119,Z 147.2,A -85,B 0,C 180,E1 -4590.768,E2 -4590.768} C_VEL
LIN {X 0,Y 524.069,Z 147.204,A -85,B 0,C 180,E1 -4593.075,E2 -4593.075} C_VEL
LIN {X 0,Y 524.033,Z 147.212,A -85,B 0,C 180,E1 -4596.159,E2 -4596.159} C_VEL
LIN {X 0,Y 524.001,Z 147.215,A -85,B 0,C 180,E1 -4598.484,E2 -4598.484} C_VEL
LIN {X 0,Y 524,Z 147.215,A -85,B 0,C 180,E1 -4601.74,E2 -4601.74} C_VEL
LIN {X 0,Y 523.99,Z 147.215,A -85,B 0,C 180,E1 -4605.052,E2 -4605.052} C_VEL
LIN {X 0,Y 523.961,Z 147.222,A -85,B 0,C 180,E1 -4607.969,E2 -4607.969} C_VEL
LIN {X 0,Y 523.969,Z 147.22,A -85,B 0,C 180,E1 -4610.41,E2 -4610.41} C_VEL
LIN {X 0,Y 523.914,Z 147.227,A -85,B 0,C 180,E1 -4612.893,E2 -4612.893} C_VEL
LIN {X 0,Y 523.95,Z 147.223,A -85,B 0,C 180,E1 -4615.419,E2 -4615.419} C_VEL
LIN {X 0,Y 523.967,Z 147.218,A -85,B 0,C 180,E1 -4617.999,E2 -4617.999} C_VEL
LIN {X 0,Y 523.942,Z 147.221,A -85,B 0,C 180,E1 -4620.855,E2 -4620.855} C_VEL
LIN {X 0,Y 523.956,Z 147.222,A -85,B 0,C 180,E1 -4623.735,E2 -4623.735} C_VEL
LIN {X 0,Y 523.9,Z 147.228,A -85,B 0,C 180,E1 -4626.402,E2 -4626.402} C_VEL
LIN {X 0,Y 523.92,Z 147.225,A -85,B 0,C 180,E1 -4629.085,E2 -4629.085} C_VEL
LIN {X 0,Y 523.954,Z 147.221,A -85,B 0,C 180,E1 -4632.119,E2 -4632.119} C_VEL
LIN {X 0,Y 523.954,Z 147.22,A -85,B 0,C 180,E1 -4635.309,E2 -4635.309} C_VEL
LIN {X 0,Y 523.954,Z 147.221,A -85,B 0,C 180,E1 -4638.69,E2 -4638.69} C_VEL
LIN {X 0,Y 523.917,Z 147.225,A -85,B 0,C 180,E1 -4641.081,E2 -4641.081} C_VEL
LIN {X 0,Y 523.922,Z 147.223,A -85,B 0,C 180,E1 -4643.828,E2 -4643.828} C_VEL
LIN {X 0,Y 523.913,Z 147.227,A -85,B 0,C 180,E1 -4646.634,E2 -4646.634} C_VEL
LIN {X 0,Y 523.955,Z 147.22,A -85,B 0,C 180,E1 -4649.356,E2 -4649.356} C_VEL
LIN {X 0,Y 523.976,Z 147.217,A -85,B 0,C 180,E1 -4652.282,E2 -4652.282} C_VEL
LIN {X 0,Y 523.952,Z 147.221,A -85,B 0,C 180,E1 -4654.582,E2 -4654.582} C_VEL
LIN {X 0,Y 523.911,Z 147.226,A -85,B 0,C 180,E1 -4657.107,E2 -4657.107} C_VEL
LIN {X 0,Y 523.98,Z 147.218,A -85,B 0,C 180,E1 -4659.866,E2 -4659.866} C_VEL
LIN {X 0,Y 523.955,Z 147.22,A -85,B 0,C 180,E1 -4662.837,E2 -4662.837} C_VEL
LIN {X 0,Y 523.976,Z 147.216,A -85,B 0,C 180,E1 -4665.236,E2 -4665.236} C_VEL
LIN {X 0,Y 524.014,Z 147.216,A -85,B 0,C 180,E1 -4668.395,E2 -4668.395} C_VEL
LIN {X 0,Y 523.991,Z 147.215,A -85,B 0,C 180,E1 -4671.516,E2 -4671.516} C_VEL
LIN {X 0,Y 524.048,Z 147.208,A -85,B 0,C 180,E1 -4673.841,E2 -4673.841} C_VEL
LIN {X 0,Y 524.073,Z 147.207,A -85,B 0,C 180,E1 -4676.926,E2 -4676.926} C_VEL
LIN {X 0,Y 524.118,Z 147.2,A -85,B 0,C 180,E1 -4680,E2 -4680} C_VEL
LIN {X 0,Y 524.072,Z 147.207,A -85,B 0,C 180,E1 -4683.075,E2 -4683.075} C_VEL
LIN {X 0,Y 524.035,Z 147.211,A -85,B 0,C 180,E1 -4686.16,E2 -4686.16} C_VEL
LIN {X 0,Y 523.989,Z 147.217,A -85,B 0,C 180,E1 -4689.262,E2 -4689.262} C_VEL
LIN {X 0,Y 524.005,Z 147.214,A -85,B 0,C 180,E1 -4691.74,E2 -4691.74} C_VEL
LIN {X 0,Y 523.995,Z 147.217,A -85,B 0,C 180,E1 -4695.052,E2 -4695.052} C_VEL
LIN {X 0,Y 523.966,Z 147.219,A -85,B 0,C 180,E1 -4697.969,E2 -4697.969} C_VEL
LIN {X 0,Y 523.975,Z 147.217,A -85,B 0,C 180,E1 -4700.41,E2 -4700.41} C_VEL
LIN {X 0,Y 523.913,Z 147.225,A -85,B 0,C 180,E1 -4702.894,E2 -4702.894} C_VEL
LIN {X 0,Y 523.955,Z 147.22,A -85,B 0,C 180,E1 -4705.419,E2 -4705.419} C_VEL
LIN {X 0,Y 523.968,Z 147.22,A -85,B 0,C 180,E1 -4707.999,E2 -4707.999} C_VEL
LIN {X 0,Y 523.947,Z 147.223,A -85,B 0,C 180,E1 -4710.855,E2 -4710.855} C_VEL
LIN {X 0,Y 523.932,Z 147.223,A -85,B 0,C 180,E1 -4713.73,E2 -4713.73} C_VEL
LIN {X 0,Y 523.906,Z 147.226,A -85,B 0,C 180,E1 -4716.402,E2 -4716.402} C_VEL
LIN {X 0,Y 523.922,Z 147.227,A -85,B 0,C 180,E1 -4719.085,E2 -4719.085} C_VEL
LIN {X 0,Y 523.954,Z 147.219,A -85,B 0,C 180,E1 -4722.119,E2 -4722.119} C_VEL
LIN {X 0,Y 523.953,Z 147.22,A -85,B 0,C 180,E1 -4725.31,E2 -4725.31} C_VEL
LIN {X 0,Y 523.958,Z 147.22,A -85,B 0,C 180,E1 -4728.69,E2 -4728.69} C_VEL
LIN {X 0,Y 523.947,Z 147.379,A -85,B 0,C 180,E1 -4731.472,E2 -4731.472} C_VEL
LIN {X 0,Y 525.056,Z 153.716,A -85,B 0,C 180,E1 -4733.917,E2 -4733.917} C_VEL
LIN {X 0,Y 525.047,Z 159.957,A -85,B 0,C 180,E1 -4736.089,E2 -4736.089} C_VEL
LIN {X 0,Y 524.826,Z 168.506,A -85,B 0,C 180,E1 -4738.985,E2 -4738.985} C_VEL
LIN {X 0,Y 524.55,Z 178.082,A -85,B 0,C 180,E1 -4742.163,E2 -4742.163} C_VEL
LIN {X 0,Y 524.316,Z 186.958,A -85,B 0,C 180,E1 -4745.025,E2 -4745.025} C_VEL
LIN {X 0,Y 524.126,Z 196.225,A -85,B 0,C 180,E1 -4747.948,E2 -4747.948} C_VEL
LIN {X 0,Y 523.926,Z 205.492,A -85,B 0,C 180,E1 -4750.813,E2 -4750.813} C_VEL
LIN {X 0,Y 523.762,Z 214.76,A -85,B 0,C 180,E1 -4753.633,E2 -4753.633} C_VEL
LIN {X 0,Y 523.644,Z 223.736,A -85,B 0,C 180,E1 -4756.286,E2 -4756.286} C_VEL
LIN {X 0,Y 525.416,Z 235.271,A -85,B 0,C 180,E1 -4756.586,E2 -4756.586} C_VEL
LIN {X 0,Y 525.205,Z 247.773,A -85,B 0,C 180,E1 -4756.999,E2 -4756.999} C_VEL
LIN {X 0,Y 524.928,Z 259.412,A -85,B 0,C 180,E1 -4757.532,E2 -4757.532} C_VEL
LIN {X 0,Y 524.674,Z 270.669,A -85,B 0,C 180,E1 -4758.207,E2 -4758.207} C_VEL
LIN {X 0,Y 524.377,Z 282.262,A -85,B 0,C 180,E1 -4759.087,E2 -4759.087} C_VEL
LIN {X 0,Y 524.095,Z 291.54,A -85,B 0,C 180,E1 -4759.961,E2 -4759.961} C_VEL
LIN {X 0,Y 523.896,Z 299.992,A -85,B 0,C 180,E1 -4760.931,E2 -4760.931} C_VEL
LIN {X 0,Y 523.688,Z 308.238,A -85,B 0,C 180,E1 -4762.094,E2 -4762.094} C_VEL
LIN {X 0,Y 523.575,Z 313.869,A -85,B 0,C 180,E1 -4763.061,E2 -4763.061} C_VEL
LIN {X 0,Y 523.544,Z 319.366,A -85,B 0,C 180,E1 -4764.222,E2 -4764.222} C_VEL
LIN {X 0,Y 523.361,Z 323.678,A -85,B 0,C 180,E1 -4765.379,E2 -4765.379} C_VEL
LIN {X 0,Y 523.443,Z 325.958,A -85,B 0,C 180,E1 -4766.151,E2 -4766.151} C_VEL
LIN {X 0,Y 523.368,Z 327.808,A -85,B 0,C 180,E1 -4766.921,E2 -4766.921} C_VEL
LIN {X 0,Y 523.335,Z 329.197,A -85,B 0,C 180,E1 -4767.691,E2 -4767.691} C_VEL
LIN {X 0,Y 523.25,Z 330.785,A -85,B 0,C 180,E1 -4769.231,E2 -4769.231} C_VEL
LIN {X 0,Y 523.246,Z 331,A -85,B 0,C 180,E1 -4770,E2 -4770} C_VEL
LIN {X 0,Y 523.275,Z 330.186,A -85,B 0,C 180,E1 -4771.539,E2 -4771.539} C_VEL
LIN {X 0,Y 523.335,Z 329.198,A -85,B 0,C 180,E1 -4772.309,E2 -4772.309} C_VEL
LIN {X 0,Y 523.368,Z 327.81,A -85,B 0,C 180,E1 -4773.079,E2 -4773.079} C_VEL
LIN {X 0,Y 523.442,Z 324.895,A -85,B 0,C 180,E1 -4774.235,E2 -4774.235} C_VEL
LIN {X 0,Y 523.464,Z 320.948,A -85,B 0,C 180,E1 -4775.393,E2 -4775.393} C_VEL
LIN {X 0,Y 523.523,Z 315.729,A -85,B 0,C 180,E1 -4776.58,E2 -4776.58} C_VEL
LIN {X 0,Y 523.665,Z 309.467,A -85,B 0,C 180,E1 -4777.713,E2 -4777.713} C_VEL
LIN {X 0,Y 523.857,Z 301.477,A -85,B 0,C 180,E1 -4778.875,E2 -4778.875} C_VEL
LIN {X 0,Y 524.086,Z 293.334,A -85,B 0,C 180,E1 -4779.845,E2 -4779.845} C_VEL
LIN {X 0,Y 524.359,Z 283.398,A -85,B 0,C 180,E1 -4780.815,E2 -4780.815} C_VEL
LIN {X 0,Y 524.63,Z 272.242,A -85,B 0,C 180,E1 -4781.685,E2 -4781.685} C_VEL
LIN {X 0,Y 524.848,Z 261.173,A -85,B 0,C 180,E1 -4782.372,E2 -4782.372} C_VEL
LIN {X 0,Y 525.169,Z 248.974,A -85,B 0,C 180,E1 -4782.953,E2 -4782.953} C_VEL
LIN {X 0,Y 525.382,Z 236.169,A -85,B 0,C 180,E1 -4783.391,E2 -4783.391} C_VEL
LIN {X 0,Y 524.75,Z 230.357,A -85,B 0,C 180,E1 -4783.555,E2 -4783.555} C_VEL
LIN {X 0,Y 523.633,Z 223.53,A -85,B 0,C 180,E1 -4783.733,E2 -4783.733} C_VEL
LIN {X 0,Y 523.762,Z 214.759,A -85,B 0,C 180,E1 -4786.367,E2 -4786.367} C_VEL
LIN {X 0,Y 523.927,Z 205.491,A -85,B 0,C 180,E1 -4789.187,E2 -4789.187} C_VEL
LIN {X 0,Y 524.13,Z 195.437,A -85,B 0,C 180,E1 -4792.299,E2 -4792.299} C_VEL
LIN {X 0,Y 524.354,Z 185.633,A -85,B 0,C 180,E1 -4795.398,E2 -4795.398} C_VEL
LIN {X 0,Y 524.609,Z 176.366,A -85,B 0,C 180,E1 -4798.397,E2 -4798.397} C_VEL
LIN {X 0,Y 524.824,Z 166.964,A -85,B 0,C 180,E1 -4801.484,E2 -4801.484} C_VEL
LIN {X 0,Y 525.052,Z 158.874,A -85,B 0,C 180,E1 -4804.207,E2 -4804.207} C_VEL
LIN {X 0,Y 525.03,Z 153.608,A -85,B 0,C 180,E1 -4806.085,E2 -4806.085} C_VEL
LIN {X 0,Y 523.941,Z 147.224,A -85,B 0,C 180,E1 -4808.631,E2 -4808.631} C_VEL
LIN {X 0,Y 523.963,Z 147.223,A -85,B 0,C 180,E1 -4811.311,E2 -4811.311} C_VEL
LIN {X 0,Y 523.961,Z 147.221,A -85,B 0,C 180,E1 -4814.691,E2 -4814.691} C_VEL
LIN {X 0,Y 523.958,Z 147.222,A -85,B 0,C 180,E1 -4817.881,E2 -4817.881} C_VEL
LIN {X 0,Y 523.926,Z 147.225,A -85,B 0,C 180,E1 -4820.915,E2 -4820.915} C_VEL
LIN {X 0,Y 523.905,Z 147.227,A -85,B 0,C 180,E1 -4823.825,E2 -4823.825} C_VEL
LIN {X 0,Y 523.947,Z 147.222,A -85,B 0,C 180,E1 -4826.636,E2 -4826.636} C_VEL
LIN {X 0,Y 523.961,Z 147.221,A -85,B 0,C 180,E1 -4829.356,E2 -4829.356} C_VEL
LIN {X 0,Y 523.984,Z 147.219,A -85,B 0,C 180,E1 -4832.281,E2 -4832.281} C_VEL
LIN {X 0,Y 523.958,Z 147.221,A -85,B 0,C 180,E1 -4834.581,E2 -4834.581} C_VEL
LIN {X 0,Y 523.916,Z 147.226,A -85,B 0,C 180,E1 -4837.106,E2 -4837.106} C_VEL
LIN {X 0,Y 523.984,Z 147.216,A -85,B 0,C 180,E1 -4839.866,E2 -4839.866} C_VEL
LIN {X 0,Y 523.959,Z 147.22,A -85,B 0,C 180,E1 -4842.837,E2 -4842.837} C_VEL
LIN {X 0,Y 523.982,Z 147.217,A -85,B 0,C 180,E1 -4845.235,E2 -4845.235} C_VEL
LIN {X 0,Y 524.018,Z 147.214,A -85,B 0,C 180,E1 -4848.394,E2 -4848.394} C_VEL
LIN {X 0,Y 524.008,Z 147.216,A -85,B 0,C 180,E1 -4851.516,E2 -4851.516} C_VEL
LIN {X 0,Y 524.087,Z 147.207,A -85,B 0,C 180,E1 -4854.613,E2 -4854.613} C_VEL
LIN {X 0,Y 524.117,Z 147.202,A -85,B 0,C 180,E1 -4857.694,E2 -4857.694} C_VEL
LIN {X 0,Y 524.128,Z 147.2,A -85,B 0,C 180,E1 -4860.768,E2 -4860.768} C_VEL
LIN {X 0,Y 524.075,Z 147.206,A -85,B 0,C 180,E1 -4863.074,E2 -4863.074} C_VEL
LIN {X 0,Y 524.049,Z 147.211,A -85,B 0,C 180,E1 -4866.159,E2 -4866.159} C_VEL
LIN {X 0,Y 523.998,Z 147.217,A -85,B 0,C 180,E1 -4868.484,E2 -4868.484} C_VEL
LIN {X 0,Y 523.802,Z 147.244,A -85,B 0,C 180,E1 -4870.826,E2 -4870.826} C_VEL
LIN {X 0,Y 523.765,Z 147.609,A -85,B 0,C 180,E1 -4871.611,E2 -4871.611} C_VEL
LIN {X 0,Y 523.716,Z 151.361,A -85,B 0,C 180,E1 -4874.937,E2 -4874.937} C_VEL
LIN {X 0,Y 523.619,Z 154.775,A -85,B 0,C 180,E1 -4877.981,E2 -4877.981} C_VEL
LIN {X 0,Y 523.545,Z 157.462,A -85,B 0,C 180,E1 -4880.427,E2 -4880.427} C_VEL
LIN {X 0,Y 523.5,Z 160.255,A -85,B 0,C 180,E1 -4882.912,E2 -4882.912} C_VEL
LIN {X 0,Y 523.522,Z 163.602,A -85,B 0,C 180,E1 -4885.915,E2 -4885.915} C_VEL
LIN {X 0,Y 523.473,Z 166.954,A -85,B 0,C 180,E1 -4888.902,E2 -4888.902} C_VEL
LIN {X 0,Y 523.461,Z 169.796,A -85,B 0,C 180,E1 -4891.407,E2 -4891.407} C_VEL
LIN {X 0,Y 525.357,Z 179.22,A -85,B 0,C 180,E1 -4891.701,E2 -4891.701} C_VEL
LIN {X 0,Y 525.237,Z 191.357,A -85,B 0,C 180,E1 -4892.132,E2 -4892.132} C_VEL
LIN {X 0,Y 524.95,Z 202.203,A -85,B 0,C 180,E1 -4892.648,E2 -4892.648} C_VEL
LIN {X 0,Y 524.672,Z 214.365,A -85,B 0,C 180,E1 -4893.401,E2 -4893.401} C_VEL
LIN {X 0,Y 524.481,Z 225.106,A -85,B 0,C 180,E1 -4894.249,E2 -4894.249} C_VEL
LIN {X 0,Y 524.198,Z 234.842,A -85,B 0,C 180,E1 -4895.205,E2 -4895.205} C_VEL
LIN {X 0,Y 523.95,Z 242.914,A -85,B 0,C 180,E1 -4896.17,E2 -4896.17} C_VEL
LIN {X 0,Y 523.749,Z 251.243,A -85,B 0,C 180,E1 -4897.396,E2 -4897.396} C_VEL
LIN {X 0,Y 523.635,Z 257.207,A -85,B 0,C 180,E1 -4898.494,E2 -4898.494} C_VEL
LIN {X 0,Y 523.519,Z 261.817,A -85,B 0,C 180,E1 -4899.545,E2 -4899.545} C_VEL
LIN {X 0,Y 522.827,Z 264.132,A -85,B 0,C 180,E1 -4900.136,E2 -4900.136} C_VEL
LIN {X 0,Y 519.892,Z 267.377,A -85,B 0,C 180,E1 -4901.116,E2 -4901.116} C_VEL
LIN {X 0,Y 517.42,Z 269.408,A -85,B 0,C 180,E1 -4901.924,E2 -4901.924} C_VEL
LIN {X 0,Y 516.359,Z 270.607,A -85,B 0,C 180,E1 -4902.558,E2 -4902.558} C_VEL
LIN {X 0,Y 516.274,Z 270.923,A -85,B 0,C 180,E1 -4902.775,E2 -4902.775} C_VEL
LIN {X 0,Y 516.243,Z 272.211,A -85,B 0,C 180,E1 -4903.971,E2 -4903.971} C_VEL
LIN {X 0,Y 516.241,Z 272.591,A -85,B 0,C 180,E1 -4905.065,E2 -4905.065} C_VEL
LIN {X 0,Y 516.241,Z 272.153,A -85,B 0,C 180,E1 -4906.18,E2 -4906.18} C_VEL
LIN {X 0,Y 516.267,Z 270.882,A -85,B 0,C 180,E1 -4907.316,E2 -4907.316} C_VEL
LIN {X 0,Y 516.33,Z 268.715,A -85,B 0,C 180,E1 -4908.471,E2 -4908.471} C_VEL
LIN {X 0,Y 516.373,Z 265.524,A -85,B 0,C 180,E1 -4909.656,E2 -4909.656} C_VEL
LIN {X 0,Y 516.484,Z 261.173,A -85,B 0,C 180,E1 -4910.861,E2 -4910.861} C_VEL
LIN {X 0,Y 516.602,Z 255.436,A -85,B 0,C 180,E1 -4912.096,E2 -4912.096} C_VEL
LIN {X 0,Y 516.783,Z 248.022,A -85,B 0,C 180,E1 -4913.356,E2 -4913.356} C_VEL
LIN {X 0,Y 517.067,Z 239.84,A -85,B 0,C 180,E1 -4914.465,E2 -4914.465} C_VEL
LIN {X 0,Y 517.303,Z 230.399,A -85,B 0,C 180,E1 -4915.508,E2 -4915.508} C_VEL
LIN {X 0,Y 517.588,Z 220.395,A -85,B 0,C 180,E1 -4916.405,E2 -4916.405} C_VEL
LIN {X 0,Y 517.84,Z 208.613,A -85,B 0,C 180,E1 -4917.242,E2 -4917.242} C_VEL
LIN {X 0,Y 518.149,Z 196.878,A -85,B 0,C 180,E1 -4917.891,E2 -4917.891} C_VEL
LIN {X 0,Y 518.436,Z 185.455,A -85,B 0,C 180,E1 -4918.368,E2 -4918.368} C_VEL
LIN {X 0,Y 518.278,Z 178.945,A -85,B 0,C 180,E1 -4918.585,E2 -4918.585} C_VEL
LIN {X 0,Y 516.349,Z 169.786,A -85,B 0,C 180,E1 -4918.885,E2 -4918.885} C_VEL
LIN {X 0,Y 516.36,Z 165.909,A -85,B 0,C 180,E1 -4922.213,E2 -4922.213} C_VEL
LIN {X 0,Y 516.437,Z 163.619,A -85,B 0,C 180,E1 -4924.184,E2 -4924.184} C_VEL
LIN {X 0,Y 516.407,Z 160.672,A -85,B 0,C 180,E1 -4926.754,E2 -4926.754} C_VEL
LIN {X 0,Y 516.439,Z 156.843,A -85,B 0,C 180,E1 -4930.11,E2 -4930.11} C_VEL
LIN {X 0,Y 516.519,Z 154.029,A -85,B 0,C 180,E1 -4932.582,E2 -4932.582} C_VEL
LIN {X 0,Y 516.558,Z 150.359,A -85,B 0,C 180,E1 -4935.824,E2 -4935.824} C_VEL
LIN {X 0,Y 516.585,Z 148.551,A -85,B 0,C 180,E1 -4937.427,E2 -4937.427} C_VEL
LIN {X 0,Y 516.705,Z 148.126,A -85,B 0,C 180,E1 -4938.323,E2 -4938.323} C_VEL
LIN {X 0,Y 516.952,Z 148.093,A -85,B 0,C 180,E1 -4941.399,E2 -4941.399} C_VEL
LIN {X 0,Y 517.025,Z 148.083,A -85,B 0,C 180,E1 -4944.54,E2 -4944.54} C_VEL
LIN {X 0,Y 517.083,Z 148.079,A -85,B 0,C 180,E1 -4947.663,E2 -4947.663} C_VEL
LIN {X 0,Y 517.09,Z 148.075,A -85,B 0,C 180,E1 -4950.779,E2 -4950.779} C_VEL
